// TIA Portal project "Program Monitoring Bearing KAI 2024 (240726)" (V14)

(* hardware
DEVICE "S7-1200 station_1"  S7-1200 Station
   slot 0: "Rack_0"  S7-1200 Rack  Rack  V1.0
   slot 1: "PLC_1"  CPU 1214C DC/DC/DC  6ES7 214-1AG40-0XB0  V4.2
   slot 2: "AI 4x13BIT_1"  6ES7 231-4HD32-0XB0  V2.0
   slot 101: "CP 1243-7 LTE"  CP 1243-7 LTE  6GK7 243-7KX30-0XE0  V3.0
      slot 0: "Telecontrol server"  Partner
      slot 0: "Inter-station communication"  Partner
DEVICE "PC-System_1"  SIMATIC PC station
   slot 0: "SIMATIC PC station"  Rail  SIMATIC PC-Station  V1.0
      slot 125: "Stationmanager"  Station_Manager  V6.0.4
   slot 1: "HMI_RT_1"  WinCC RT Advanced  6AV2 104-0xxxx-xxxx  14.0.1.0
      slot 33792: "Host interface"  Host interface
   slot 2: "IE general_1"  IE General  IE_CP  V8.2.0
*)

// ===== PLC "PLC_1"  CPU 1214C DC/DC/DC =====

VAR_GLOBAL   // PLC tag table "Default tag table"
   "prox_a1" AT %I0.0 : Bool;
   "prox_b1" AT %I0.1 : Bool;
   "Q1-1" AT %M0.0 : Bool;   // utk ngasi trigger biar sensor suhu ngebaca
   "Q2-1" AT %M0.1 : Bool;   // utk ngasi trigger biar sensor suhu ngebaca
   "du_a" AT %M0.2 : Bool;
   "dd_b" AT %M0.3 : Bool;
   "counter" AT %M0.6 : Bool;
   "pemutus" AT %M0.7 : Bool;
   "ProxA+" AT %M1.0 : Bool;
   "ProxB-" AT %M1.1 : Bool;
   "reset" AT %M1.2 : Bool;
   "Clock_Byte" AT %MB10 : Byte;
   "Clock_10Hz" AT %M10.0 : Bool;
   "Clock_5Hz" AT %M10.1 : Bool;
   "Clock_2.5Hz" AT %M10.2 : Bool;
   "Clock_2Hz" AT %M10.3 : Bool;
   "Clock_1.25Hz" AT %M10.4 : Bool;
   "Clock_1Hz" AT %M10.5 : Bool;
   "Clock_0.625Hz" AT %M10.6 : Bool;
   "Clock_0.5Hz" AT %M10.7 : Bool;
   "System_Byte" AT %MB100 : Byte;
   "FirstScan" AT %M100.0 : Bool;
   "DiagStatusUpdate" AT %M100.1 : Bool;
   "AlwaysTRUE" AT %M100.2 : Bool;
   "AlwaysFALSE" AT %M100.3 : Bool;
   "led1" AT %Q0.2 : Bool;
   "led2" AT %Q0.3 : Bool;
   "led3" AT %Q0.4 : Bool;
   "led4" AT %Q0.5 : Bool;
   "led5" AT %Q0.6 : Bool;
   "led6" AT %Q0.7 : Bool;
   "Actual_Step" AT %MW2 : Int;
   "ganjil" AT %M4.0 : Bool;
   "pemutus2" AT %M4.1 : Bool;
   "Q1--2" AT %M2.0 : Bool;   // dipake if nanti sensor suhu ny jd 2 buah (utk datang kanan)
   "Q2-2" AT %M2.1 : Bool;   // dipake if nanti sensor suhu ny jd 2 buah (utk datang kiri)
   "koil timer" AT %M2.4 : Bool;
   "reset koil" AT %M2.3 : Bool;
   "Tag_2" AT %M2.5 : Bool;
   "AI_Sensor Suhu" AT %IW96 : Int;
   "AI_0_Scaled" AT %MD6 : Real;
   "PowerSensorSuhu" AT %Q0.0 : Bool;   // kalo sensor suhu ny jd 2 buah, tambahin satu lg (simpen d network2)
   "Tag_1" AT %M5.0 : Bool;
   "Tag_3" AT %M5.1 : Bool;
   "Tag_4" AT %M5.2 : Bool;
   "Tag_5" AT %M8.0 : Bool;
   "Tag_6" AT %M4.2 : Bool;
   "Tag_7" AT %M9.0 : Bool;
   "Tag_8" AT %M9.3 : Bool;
   "Tag_9" AT %M6.7 : Bool;
   "Tag_10" AT %M12.0 : Bool;
   "Tag_11" AT %MD0 : Time;
   "Tag_12" AT %M8.1 : Bool;
   "Tag_13" AT %M3.0 : Bool;
   "Tag_14" AT %M9.4 : Bool;
   "Tag_15" AT %I0.2 : Bool;
   "Tag_16" AT %M4.4 : Bool;
   "Tag_17" AT %M9.1 : Bool;
   "Tag_18" AT %M9.2 : Bool;
   "Tag_19" AT %M4.3 : Bool;
   "Tag_20" AT %MD2 : DWord;
   "Tag_21" AT %M7.2 : Bool;
   "Tag_22" AT %M3.1 : Bool;
   "Tag_23" AT %M1.3 : Bool;
   "Tag_24" AT %Q1.0 : Bool;
   "Tag_25" AT %M1.4 : Bool;
   "timer_reset" AT %M1.5 : Bool;
   "Suhu_Kanan" AT %MD10 : Real;
   "Tag_27" AT %MD11 : Real;
   "Suhu_Kiri" AT %MD12 : Real;
   "Tag_29" AT %MD13 : Real;
   "Tag_30" AT %MD14 : Real;
   "Tag_31" AT %MD15 : Real;
   "Tag_32" AT %MD16 : Real;
   "Tag_33" AT %MD20 : Real;
   "Tag_34" AT %MD21 : Real;
   "Tag_35" AT %M4.5 : Bool;
   "Tag_36" AT %M4.6 : Bool;
   "Tag_37" AT %M1.6 : Bool;
   "Tag_38" AT %M3.2 : Bool;
   "Tag_39" AT %M3.3 : Bool;
   "Tag_40" AT %M2.2 : Bool;
   "Tag_41" AT %M6.0 : Bool;
   "Tag_42" AT %M6.1 : Bool;
   "Tag_43" AT %M6.2 : Bool;
   "Tag_44" AT %M6.3 : Bool;
   "Tag_45" AT %M6.4 : Bool;
   "Tag_46" AT %M6.5 : Bool;
   "Tag_47" AT %M6.6 : Bool;
   "Tag_48" AT %M7.3 : Bool;
   "Tag_49" AT %M7.4 : Bool;
   "memoryA1" AT %M2.6 : Bool;
   "MemoryB1" AT %M2.7 : Bool;
   "Tag_26" AT %MD1 : Time;
END_VAR

DATA_BLOCK "Data_block_1"   // DB3
{ S7_Optimized_Access := 'FALSE' }
VERSION : 0.1
   VAR
      "counter" : Int;
      "identitas kereta" : String;
      counter_datasuhu : Int := 1;
      sarana : String;
      ganjil : Int := -1;
      genap : Int;
      datasuhu1 : Real;   // Kanan
      datasuhu2 : Real;   // Kiri
      rodakirike : Int;
      rodakananke : Int;
      K1 : Bool;   // Kanan
      K2 : Bool;   // Kiri
      ResetCounterDataSensor : Bool;   // Kanan
      ResetCounterDataSensor1 : Bool;   // Kiri
      ResetCounter100 : Bool;
      Reset : Bool;
      InputKecepatan : Bool;   // Kanan
      InputKecepatan1 : Bool;   // Kiri
      KecepatanKereta : Real;
      Lock_A : Bool;   // Kanan
      Lock_B : Bool;   // Kiri
      ProxB_P : Bool;
      ProxB_N : Bool;
      ProxA_N : Bool;
      ProxA_P : Bool;
      K_B : Bool;
      K_A : Bool;
      WaktuTempuhSensor : Real;
      TimeInput : Bool;
      TimerSensor : Time := T#1ms;
      TimerReset : Time := T#5m;
      datasensor1 : Real;
      datasensor2 : Real;
      data_baru1 : Array[0..99] of Real;   // Kanan
      data_baru2 : Array[0..99] of Real;   // Kiri
      data_suhu_bearing1 : Array[0..99] of Real;
      data_suhu_bearing2 : Array[0..99] of Real;
      data_suhu_bearing3 : Array[0..99] of Real;
      data_suhu_bearing4 : Array[0..99] of Real;
      data_suhu_bearing5 : Array[0..99] of Real;
      data_suhu_bearing6 : Array[0..99] of Real;
      data_suhu_bearing7 : Array[0..99] of Real;
      data_suhu_bearing8 : Array[0..99] of Real;
      data_suhu_bearing9 : Array[0..99] of Real;
      data_suhu_bearing10 : Array[0..99] of Real;
      data_suhu_bearing11 : Array[0..99] of Real;
      data_suhu_bearing12 : Array[0..99] of Real;
      data_suhu_bearing13 : Array[0..99] of Real;
      data_suhu_bearing14 : Array[0..99] of Real;
      data_suhu_bearing15 : Array[0..99] of Real;
      data_suhu_bearing16 : Array[0..99] of Real;
      data_suhu_bearing17 : Array[0..99] of Real;
      data_suhu_bearing18 : Array[0..99] of Real;
      data_suhu_bearing19 : Array[0..99] of Real;
      data_suhu_bearing20 : Array[0..99] of Real;
      data_suhu_bearing21 : Array[0..99] of Real;
      data_suhu_bearing22 : Array[0..99] of Real;
      data_suhu_bearing23 : Array[0..99] of Real;
      data_suhu_bearing24 : Array[0..99] of Real;
      data_suhu_bearing25 : Array[0..99] of Real;
      data_suhu_bearing26 : Array[0..99] of Real;
      data_suhu_bearing27 : Array[0..99] of Real;
      data_suhu_bearing28 : Array[0..99] of Real;
      data_suhu_bearing29 : Array[0..99] of Real;
      data_suhu_bearing30 : Array[0..99] of Real;
      data_suhu_bearing31 : Array[0..99] of Real;
      data_suhu_bearing32 : Array[0..99] of Real;
      data_suhu_bearing33 : Array[0..99] of Real;
      data_suhu_bearing34 : Array[0..99] of Real;
      data_suhu_bearing35 : Array[0..99] of Real;
      data_suhu_bearing36 : Array[0..99] of Real;
      data_suhu_bearing37 : Array[0..99] of Real;
      data_suhu_bearing38 : Array[0..99] of Real;
      data_suhu_bearing39 : Array[0..99] of Real;
      data_suhu_bearing40 : Array[0..99] of Real;
      data_suhu_bearing41 : Array[0..99] of Real;
      data_suhu_bearing42 : Array[0..99] of Real;
      data_suhu_bearing43 : Array[0..99] of Real;
      data_suhu_bearing44 : Array[0..99] of Real;
      data_suhu_bearing45 : Array[0..99] of Real;
      data_suhu_bearing46 : Array[0..99] of Real;
      data_suhu_bearing47 : Array[0..99] of Real;
      data_suhu_bearing48 : Array[0..99] of Real;
      data_suhu_bearing49 : Array[0..99] of Real;
      data_suhu_bearing50 : Array[0..99] of Real;
      data_lama1 : Real;   // Kanan
      data_lama2 : Real;   // Kiri
      dataroda1 : Array[0..49] of Real;   // Kanan
      dataroda2 : Array[0..49] of Real;   // Kiri
      data_0 : Array[0..99] of Real;
      Reset_data_baru1 : Bool;
      counter_sensorA : Int;
      counter_sensorB : Int;
      counterAK1 : Int;
      counterBK1 : Int;
      counterAnotB : Int;
      counterABnot : Int;
      counter_2 : Int;
      counter_1 : Int;
      K10 : Bool;
      counterk1 : Int;
      counterAB : Int;
   END_VAR
BEGIN
END_DATA_BLOCK

// folder: System blocks/Program resources

DATA_BLOCK "IEC_Counter_0_DB_8"   // DB1
{ S7_Optimized_Access := 'TRUE' }
AUTHOR : Simatic
FAMILY : IEC
NAME : CNTR
VERSION : 1.0
// stored: InstanceOfName IEC_COUNTER
"IEC_COUNTER"
BEGIN
END_DATA_BLOCK

DATA_BLOCK "IEC_Timer_0_DB"   // DB2
{ S7_Optimized_Access := 'TRUE' }
AUTHOR : Simatic
FAMILY : IEC
NAME : IEC_TMR
VERSION : 1.0
// stored: InstanceOfName IEC_TIMER
"IEC_TIMER"
BEGIN
END_DATA_BLOCK

DATA_BLOCK "IEC_Counter_0_DB"   // DB4
{ S7_Optimized_Access := 'TRUE' }
AUTHOR : Simatic
FAMILY : IEC
NAME : CNTR
VERSION : 1.0
// stored: InstanceOfName IEC_COUNTER
"IEC_COUNTER"
BEGIN
END_DATA_BLOCK

DATA_BLOCK "IEC_Timer_0_DB_2"   // DB5
{ S7_Optimized_Access := 'TRUE' }
AUTHOR : Simatic
FAMILY : IEC
NAME : IEC_TMR
VERSION : 1.0
// stored: InstanceOfName IEC_TIMER
"IEC_TIMER"
BEGIN
END_DATA_BLOCK

DATA_BLOCK "IEC_Timer_0_DB_1"   // DB6
{ S7_Optimized_Access := 'TRUE' }
AUTHOR : Simatic
FAMILY : IEC
NAME : IEC_TMR
VERSION : 1.0
// stored: InstanceOfName IEC_TIMER
"IEC_TIMER"
BEGIN
END_DATA_BLOCK

DATA_BLOCK "IEC_Timer_0_DB_4"   // DB7
{ S7_Optimized_Access := 'TRUE' }
AUTHOR : Simatic
FAMILY : IEC
NAME : IEC_TMR
VERSION : 1.0
// stored: InstanceOfName IEC_TIMER
"IEC_TIMER"
BEGIN
END_DATA_BLOCK

DATA_BLOCK "IEC_Timer_0_DB_3"   // DB8
{ S7_Optimized_Access := 'TRUE' }
AUTHOR : Simatic
FAMILY : IEC
NAME : IEC_TMR
VERSION : 1.0
// stored: InstanceOfName IEC_TIMER
"IEC_TIMER"
BEGIN
END_DATA_BLOCK

DATA_BLOCK "IEC_Timer_0_DB_5"   // DB9
{ S7_Optimized_Access := 'TRUE' }
AUTHOR : Simatic
FAMILY : IEC
NAME : IEC_TMR
VERSION : 1.0
// stored: InstanceOfName IEC_TIMER
"IEC_TIMER"
BEGIN
END_DATA_BLOCK

DATA_BLOCK "IEC_Counter_0_DB_1"   // DB10
{ S7_Optimized_Access := 'TRUE' }
AUTHOR : Simatic
FAMILY : IEC
NAME : CNTR
VERSION : 1.0
// stored: InstanceOfName IEC_COUNTER
"IEC_COUNTER"
BEGIN
END_DATA_BLOCK

DATA_BLOCK "IEC_Timer_0_DB_7"   // DB11
{ S7_Optimized_Access := 'TRUE' }
AUTHOR : Simatic
FAMILY : IEC
NAME : IEC_TMR
VERSION : 1.0
// stored: InstanceOfName IEC_TIMER
"IEC_TIMER"
BEGIN
END_DATA_BLOCK

DATA_BLOCK "IEC_Timer_0_DB_8"   // DB12
{ S7_Optimized_Access := 'TRUE' }
AUTHOR : Simatic
FAMILY : IEC
NAME : IEC_TMR
VERSION : 1.0
// stored: InstanceOfName IEC_TIMER
"IEC_TIMER"
BEGIN
END_DATA_BLOCK

DATA_BLOCK "IEC_Timer_0_DB_9"   // DB13
{ S7_Optimized_Access := 'TRUE' }
AUTHOR : Simatic
FAMILY : IEC
NAME : IEC_TMR
VERSION : 1.0
// stored: InstanceOfName IEC_TIMER
"IEC_TIMER"
BEGIN
END_DATA_BLOCK

DATA_BLOCK "IEC_Timer_0_DB_10"   // DB14
{ S7_Optimized_Access := 'TRUE' }
AUTHOR : Simatic
FAMILY : IEC
NAME : IEC_TMR
VERSION : 1.0
// stored: InstanceOfName IEC_TIMER
"IEC_TIMER"
BEGIN
END_DATA_BLOCK

DATA_BLOCK "IEC_Timer_0_DB_11"   // DB15
{ S7_Optimized_Access := 'TRUE' }
AUTHOR : Simatic
FAMILY : IEC
NAME : IEC_TMR
VERSION : 1.0
// stored: InstanceOfName IEC_TIMER
"IEC_TIMER"
BEGIN
END_DATA_BLOCK

DATA_BLOCK "IEC_Counter_0_DB_2"   // DB17
{ S7_Optimized_Access := 'TRUE' }
AUTHOR : Simatic
FAMILY : IEC
NAME : CNTR
VERSION : 1.0
// stored: InstanceOfName IEC_COUNTER
"IEC_COUNTER"
BEGIN
END_DATA_BLOCK

DATA_BLOCK "IEC_Counter_0_DB_3"   // DB18
{ S7_Optimized_Access := 'TRUE' }
AUTHOR : Simatic
FAMILY : IEC
NAME : CNTR
VERSION : 1.0
// stored: InstanceOfName IEC_COUNTER
"IEC_COUNTER"
BEGIN
END_DATA_BLOCK

DATA_BLOCK "IEC_Counter_0_DB_4"   // DB19
{ S7_Optimized_Access := 'TRUE' }
AUTHOR : Simatic
FAMILY : IEC
NAME : CNTR
VERSION : 1.0
// stored: InstanceOfName IEC_COUNTER
"IEC_COUNTER"
BEGIN
END_DATA_BLOCK

DATA_BLOCK "IEC_Counter_0_DB_5"   // DB20
{ S7_Optimized_Access := 'TRUE' }
AUTHOR : Simatic
FAMILY : IEC
NAME : CNTR
VERSION : 1.0
// stored: InstanceOfName IEC_COUNTER
"IEC_COUNTER"
BEGIN
END_DATA_BLOCK

DATA_BLOCK "IEC_Counter_0_DB_6"   // DB21
{ S7_Optimized_Access := 'TRUE' }
AUTHOR : Simatic
FAMILY : IEC
NAME : CNTR
VERSION : 1.0
// stored: InstanceOfName IEC_COUNTER
"IEC_COUNTER"
BEGIN
END_DATA_BLOCK

DATA_BLOCK "IEC_Counter_0_DB_7"   // DB22
{ S7_Optimized_Access := 'TRUE' }
AUTHOR : Simatic
FAMILY : IEC
NAME : CNTR
VERSION : 1.0
// stored: InstanceOfName IEC_COUNTER
"IEC_COUNTER"
BEGIN
END_DATA_BLOCK

DATA_BLOCK "IEC_Counter_0_DB_11"   // DB23
{ S7_Optimized_Access := 'TRUE' }
AUTHOR : Simatic
FAMILY : IEC
NAME : CNTR
VERSION : 1.0
// stored: InstanceOfName IEC_COUNTER
"IEC_COUNTER"
BEGIN
END_DATA_BLOCK

DATA_BLOCK "IEC_Timer_0_DB_6"   // DB24
{ S7_Optimized_Access := 'TRUE' }
AUTHOR : Simatic
FAMILY : IEC
NAME : IEC_TMR
VERSION : 1.0
// stored: InstanceOfName IEC_TIMER
"IEC_TIMER"
BEGIN
END_DATA_BLOCK

DATA_BLOCK "IEC_Timer_0_DB_12"   // DB25
{ S7_Optimized_Access := 'TRUE' }
AUTHOR : Simatic
FAMILY : IEC
NAME : IEC_TMR
VERSION : 1.0
// stored: InstanceOfName IEC_TIMER
"IEC_TIMER"
BEGIN
END_DATA_BLOCK

// folder: (top level)

FUNCTION "Block_1" : Void   // FC1, LAD
{ S7_Optimized_Access := 'TRUE' }
VERSION : 0.1
   VAR_INPUT
      "analog input suhu" : Int;
      lower : Real;
      upper : Real;
   END_VAR
   VAR_OUTPUT
      "Scaled Output Suhu" : Real;
   END_VAR
   VAR_TEMP
      Temp1 : Real;   // temporary data
   END_VAR
BEGIN

REGION Network 1
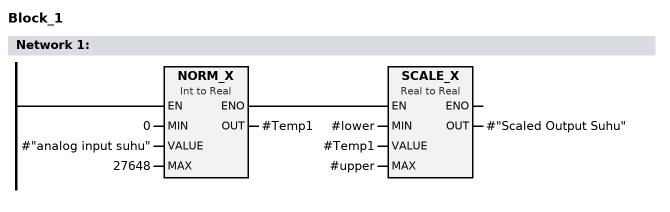
   RUNG wire#powerrail
      { S7_Templates := "[SrcType := Int, DestType := Real]" } Normalize(min := 0, value := #"analog input suhu", max := 27648, out => #Temp1)
      { S7_Templates := "[SrcType := Real, DestType := Real]" } Scale(min := #lower, value := #Temp1, max := #upper, out => #"Scaled Output Suhu")
   END_RUNG
   // the same network as SCL:
   #Temp1 := NORM_X(MIN := 0, VALUE := #"analog input suhu", MAX := 27648);
   #"Scaled Output Suhu" := SCALE_X(MIN := #lower, VALUE := #Temp1, MAX := #upper);
END_REGION
END_FUNCTION

ORGANIZATION_BLOCK "Program Datang Kiri"   // OB1, LAD, ProgramCycle
TITLE = Datang Kiri
{ S7_Optimized_Access := 'TRUE' }
VERSION : 0.1
   VAR_INPUT
      Initial_Call : Bool;   // Initial call of this OB
      Remanence : Bool;   // =True, if remanent data are available
   END_VAR
   VAR CONSTANT
      initial_step : Int;
      step_led1 : Int := 1;
      step_led2 : Int := 2;
      step_led3 : Int := 3;
      step_led4 : Int := 4;
      step_led5 : Int := 5;
      step_led6 : Int := 6;
   END_VAR
   VAR_TEMP   // added for the SCL form of the ladder/FBD networks
      _w1 : Bool;
      _w2 : Bool;
      _w3 : Bool;
      _w4 : Bool;
      _w5 : Bool;
      _w6 : Bool;
      _w7 : Bool;
      _w8 : Bool;
      _w9 : Bool;
      _w10 : Bool;
      _w11 : Bool;
      _w12 : Bool;
      _w13 : Bool;
      _w14 : Bool;
      _w15 : Bool;
      _w16 : Bool;
      _w17 : Bool;
      _w18 : Bool;
      _w19 : Bool;
      _w20 : Bool;
      _w21 : Bool;
      _w22 : Bool;
      _w23 : Bool;
      _w24 : Bool;
      _w25 : Bool;
      _w26 : Bool;
      _w27 : Bool;
      _w28 : Bool;
      _w29 : Bool;
      _w30 : Bool;
      _w31 : Bool;
      _w32 : Bool;
      _w33 : Bool;
      _w34 : Bool;
      _w35 : Bool;
      _w36 : Bool;
      _w37 : Bool;
      _w38 : Bool;
      _w39 : Bool;
      _w40 : Bool;
      _w41 : Bool;
      _w42 : Bool;
      _w43 : Bool;
      _w44 : Bool;
      _w45 : Bool;
      _w46 : Bool;
      _w47 : Bool;
      _w48 : Bool;
      _w49 : Bool;
      _w50 : Bool;
   END_VAR
BEGIN

REGION Network 1: Koil Mengukur kecepatan kereta (kiri ke kanan)
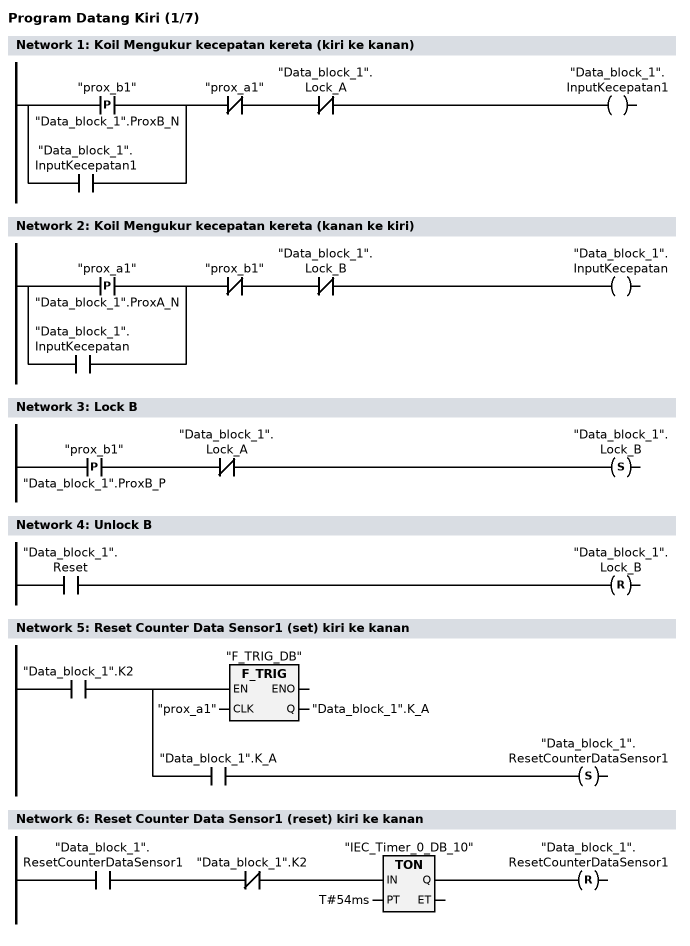
   RUNG wire#powerrail
      P_Contact(operand := "prox_b1", bit := "Data_block_1".ProxB_N)
      wire#w1
      I_Contact( "prox_a1" )
      I_Contact( "Data_block_1".Lock_A )
      Coil( "Data_block_1".InputKecepatan1 )
   END_RUNG
   RUNG wire#powerrail
      Contact( "Data_block_1".InputKecepatan1 )
   END_RUNG wire#w1
   // the same network as SCL:
   #_w1 := "prox_b1" AND NOT "Data_block_1".ProxB_N;   // rising edge of "prox_b1"
   "Data_block_1".ProxB_N := "prox_b1";
   "Data_block_1".InputKecepatan1 := (#_w1 OR "Data_block_1".InputKecepatan1) AND NOT "prox_a1" AND NOT "Data_block_1".Lock_A;
END_REGION

REGION Network 2: Koil Mengukur kecepatan kereta (kanan ke kiri)
   RUNG wire#powerrail
      P_Contact(operand := "prox_a1", bit := "Data_block_1".ProxA_N)
      wire#w1
      I_Contact( "prox_b1" )
      I_Contact( "Data_block_1".Lock_B )
      Coil( "Data_block_1".InputKecepatan )
   END_RUNG
   RUNG wire#powerrail
      Contact( "Data_block_1".InputKecepatan )
   END_RUNG wire#w1
   // the same network as SCL:
   #_w1 := "prox_a1" AND NOT "Data_block_1".ProxA_N;   // rising edge of "prox_a1"
   "Data_block_1".ProxA_N := "prox_a1";
   "Data_block_1".InputKecepatan := (#_w1 OR "Data_block_1".InputKecepatan) AND NOT "prox_b1" AND NOT "Data_block_1".Lock_B;
END_REGION

REGION Network 3: Lock B
   RUNG wire#powerrail
      P_Contact(operand := "prox_b1", bit := "Data_block_1".ProxB_P)
      I_Contact( "Data_block_1".Lock_A )
      S_Coil( "Data_block_1".Lock_B )
   END_RUNG
   // the same network as SCL:
   #_w1 := "prox_b1" AND NOT "Data_block_1".ProxB_P;   // rising edge of "prox_b1"
   "Data_block_1".ProxB_P := "prox_b1";
   IF #_w1 AND NOT "Data_block_1".Lock_A THEN "Data_block_1".Lock_B := TRUE; END_IF;
END_REGION

REGION Network 4: Unlock B
   RUNG wire#powerrail
      Contact( "Data_block_1".Reset )
      R_Coil( "Data_block_1".Lock_B )
   END_RUNG
   // the same network as SCL:
   IF "Data_block_1".Reset THEN "Data_block_1".Lock_B := FALSE; END_IF;
END_REGION

REGION Network 5: Reset Counter Data Sensor1 (set) kiri ke kanan
   IF "Data_block_1".K2 THEN
       "F_TRIG_DB"(CLK := "prox_a1", Q => "Data_block_1".K_A);   // F_TRIG
   END_IF;
   IF "Data_block_1".K2 AND "Data_block_1".K_A THEN "Data_block_1".ResetCounterDataSensor1 := TRUE; END_IF;
END_REGION

REGION Network 6: Reset Counter Data Sensor1 (reset) kiri ke kanan
   "IEC_Timer_0_DB_10".TON(IN := "Data_block_1".ResetCounterDataSensor1 AND NOT "Data_block_1".K2, PT := T#54ms);
   IF "IEC_Timer_0_DB_10".Q THEN "Data_block_1".ResetCounterDataSensor1 := FALSE; END_IF;
END_REGION

REGION Network 7: reset data_baru (kiri ke kanan) data_baru2
   // ketika reset aktif 
   // 
   // - maka datasuhu, array data suhu roda akan kembali 0
   // - maka counter genap kembali 0
   // - maka counter ganjil menjadi -1
   // - maka sarana akan kosong
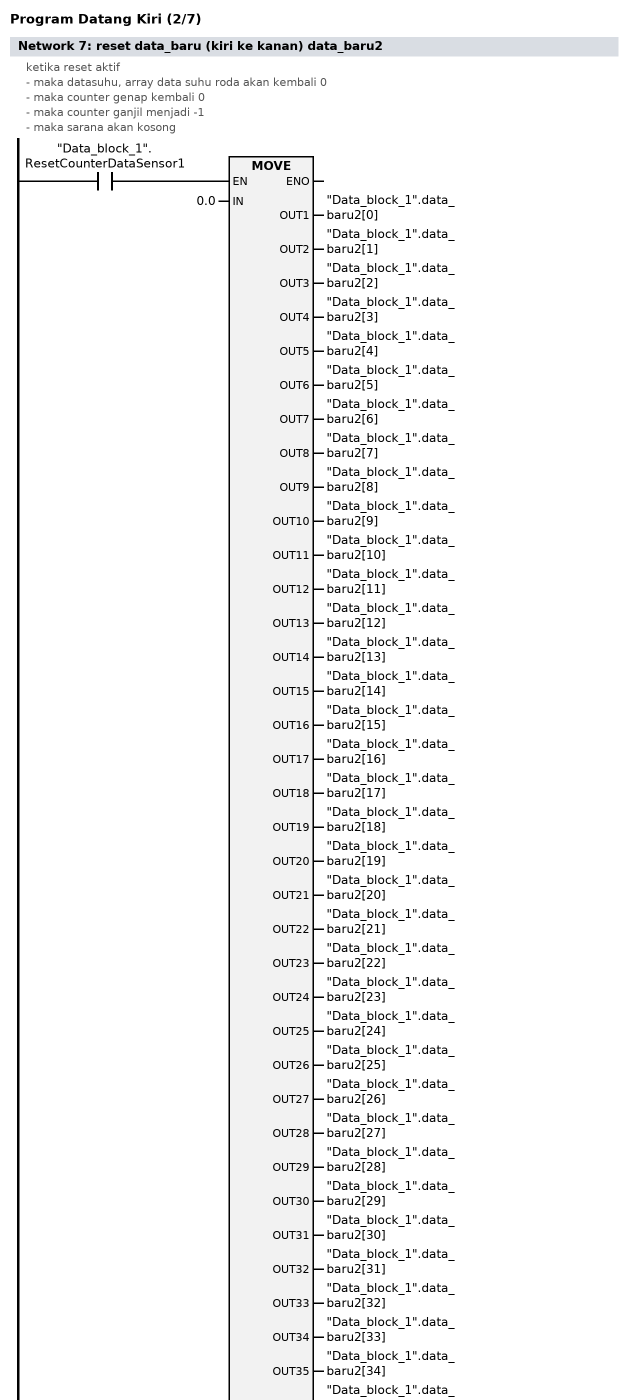
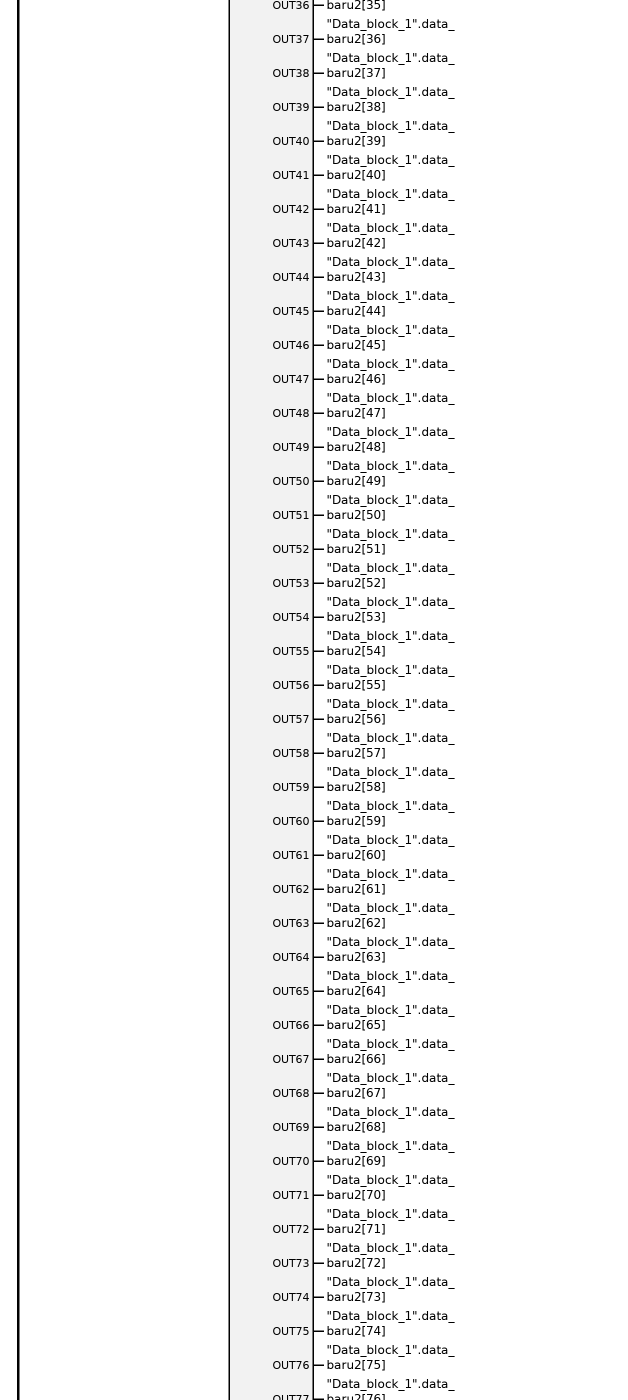
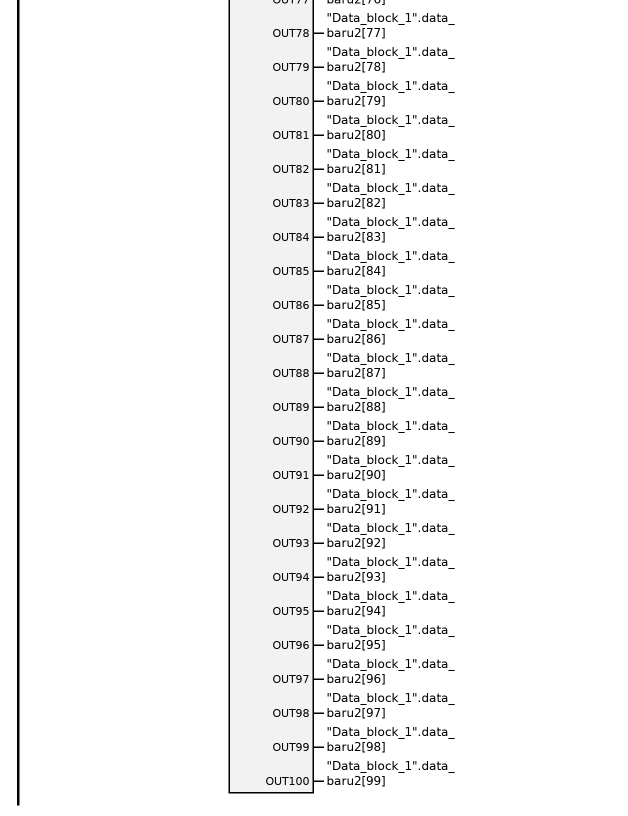
   RUNG wire#powerrail
      Contact( "Data_block_1".ResetCounterDataSensor1 )
      Move(in := 0.0, out1 => "Data_block_1".data_baru2[0], out2 => "Data_block_1".data_baru2[1], out3 => "Data_block_1".data_baru2[2], out4 => "Data_block_1".data_baru2[3], out5 => "Data_block_1".data_baru2[4], out6 => "Data_block_1".data_baru2[5], out7 => "Data_block_1".data_baru2[6], out8 => "Data_block_1".data_baru2[7], out9 => "Data_block_1".data_baru2[8], out10 => "Data_block_1".data_baru2[9], out11 => "Data_block_1".data_baru2[10], out12 => "Data_block_1".data_baru2[11], out13 => "Data_block_1".data_baru2[12], out14 => "Data_block_1".data_baru2[13], out15 => "Data_block_1".data_baru2[14], out16 => "Data_block_1".data_baru2[15], out17 => "Data_block_1".data_baru2[16], out18 => "Data_block_1".data_baru2[17], out19 => "Data_block_1".data_baru2[18], out20 => "Data_block_1".data_baru2[19], out21 => "Data_block_1".data_baru2[20], out22 => "Data_block_1".data_baru2[21], out23 => "Data_block_1".data_baru2[22], out24 => "Data_block_1".data_baru2[23], out25 => "Data_block_1".data_baru2[24], out26 => "Data_block_1".data_baru2[25], out27 => "Data_block_1".data_baru2[26], out28 => "Data_block_1".data_baru2[27], out29 => "Data_block_1".data_baru2[28], out30 => "Data_block_1".data_baru2[29], out31 => "Data_block_1".data_baru2[30], out32 => "Data_block_1".data_baru2[31], out33 => "Data_block_1".data_baru2[32], out34 => "Data_block_1".data_baru2[33], out35 => "Data_block_1".data_baru2[34], out36 => "Data_block_1".data_baru2[35], out37 => "Data_block_1".data_baru2[36], out38 => "Data_block_1".data_baru2[37], out39 => "Data_block_1".data_baru2[38], out40 => "Data_block_1".data_baru2[39], out41 => "Data_block_1".data_baru2[40], out42 => "Data_block_1".data_baru2[41], out43 => "Data_block_1".data_baru2[42], out44 => "Data_block_1".data_baru2[43], out45 => "Data_block_1".data_baru2[44], out46 => "Data_block_1".data_baru2[45], out47 => "Data_block_1".data_baru2[46], out48 => "Data_block_1".data_baru2[47], out49 => "Data_block_1".data_baru2[48], out50 => "Data_block_1".data_baru2[49], out51 => "Data_block_1".data_baru2[50], out52 => "Data_block_1".data_baru2[51], out53 => "Data_block_1".data_baru2[52], out54 => "Data_block_1".data_baru2[53], out55 => "Data_block_1".data_baru2[54], out56 => "Data_block_1".data_baru2[55], out57 => "Data_block_1".data_baru2[56], out58 => "Data_block_1".data_baru2[57], out59 => "Data_block_1".data_baru2[58], out60 => "Data_block_1".data_baru2[59], out61 => "Data_block_1".data_baru2[60], out62 => "Data_block_1".data_baru2[61], out63 => "Data_block_1".data_baru2[62], out64 => "Data_block_1".data_baru2[63], out65 => "Data_block_1".data_baru2[64], out66 => "Data_block_1".data_baru2[65], out67 => "Data_block_1".data_baru2[66], out68 => "Data_block_1".data_baru2[67], out69 => "Data_block_1".data_baru2[68], out70 => "Data_block_1".data_baru2[69], out71 => "Data_block_1".data_baru2[70], out72 => "Data_block_1".data_baru2[71], out73 => "Data_block_1".data_baru2[72], out74 => "Data_block_1".data_baru2[73], out75 => "Data_block_1".data_baru2[74], out76 => "Data_block_1".data_baru2[75], out77 => "Data_block_1".data_baru2[76], out78 => "Data_block_1".data_baru2[77], out79 => "Data_block_1".data_baru2[78], out80 => "Data_block_1".data_baru2[79], out81 => "Data_block_1".data_baru2[80], out82 => "Data_block_1".data_baru2[81], out83 => "Data_block_1".data_baru2[82], out84 => "Data_block_1".data_baru2[83], out85 => "Data_block_1".data_baru2[84], out86 => "Data_block_1".data_baru2[85], out87 => "Data_block_1".data_baru2[86], out88 => "Data_block_1".data_baru2[87], out89 => "Data_block_1".data_baru2[88], out90 => "Data_block_1".data_baru2[89], out91 => "Data_block_1".data_baru2[90], out92 => "Data_block_1".data_baru2[91], out93 => "Data_block_1".data_baru2[92], out94 => "Data_block_1".data_baru2[93], out95 => "Data_block_1".data_baru2[94], out96 => "Data_block_1".data_baru2[95], out97 => "Data_block_1".data_baru2[96], out98 => "Data_block_1".data_baru2[97], out99 => "Data_block_1".data_baru2[98], out100 => "Data_block_1".data_baru2[99])
   END_RUNG
   // the same network as SCL:
   IF "Data_block_1".ResetCounterDataSensor1 THEN
       "Data_block_1".data_baru2[0] := 0.0;
       "Data_block_1".data_baru2[1] := 0.0;
       "Data_block_1".data_baru2[2] := 0.0;
       "Data_block_1".data_baru2[3] := 0.0;
       "Data_block_1".data_baru2[4] := 0.0;
       "Data_block_1".data_baru2[5] := 0.0;
       "Data_block_1".data_baru2[6] := 0.0;
       "Data_block_1".data_baru2[7] := 0.0;
       "Data_block_1".data_baru2[8] := 0.0;
       "Data_block_1".data_baru2[9] := 0.0;
       "Data_block_1".data_baru2[10] := 0.0;
       "Data_block_1".data_baru2[11] := 0.0;
       "Data_block_1".data_baru2[12] := 0.0;
       "Data_block_1".data_baru2[13] := 0.0;
       "Data_block_1".data_baru2[14] := 0.0;
       "Data_block_1".data_baru2[15] := 0.0;
       "Data_block_1".data_baru2[16] := 0.0;
       "Data_block_1".data_baru2[17] := 0.0;
       "Data_block_1".data_baru2[18] := 0.0;
       "Data_block_1".data_baru2[19] := 0.0;
       "Data_block_1".data_baru2[20] := 0.0;
       "Data_block_1".data_baru2[21] := 0.0;
       "Data_block_1".data_baru2[22] := 0.0;
       "Data_block_1".data_baru2[23] := 0.0;
       "Data_block_1".data_baru2[24] := 0.0;
       "Data_block_1".data_baru2[25] := 0.0;
       "Data_block_1".data_baru2[26] := 0.0;
       "Data_block_1".data_baru2[27] := 0.0;
       "Data_block_1".data_baru2[28] := 0.0;
       "Data_block_1".data_baru2[29] := 0.0;
       "Data_block_1".data_baru2[30] := 0.0;
       "Data_block_1".data_baru2[31] := 0.0;
       "Data_block_1".data_baru2[32] := 0.0;
       "Data_block_1".data_baru2[33] := 0.0;
       "Data_block_1".data_baru2[34] := 0.0;
       "Data_block_1".data_baru2[35] := 0.0;
       "Data_block_1".data_baru2[36] := 0.0;
       "Data_block_1".data_baru2[37] := 0.0;
       "Data_block_1".data_baru2[38] := 0.0;
       "Data_block_1".data_baru2[39] := 0.0;
       "Data_block_1".data_baru2[40] := 0.0;
       "Data_block_1".data_baru2[41] := 0.0;
       "Data_block_1".data_baru2[42] := 0.0;
       "Data_block_1".data_baru2[43] := 0.0;
       "Data_block_1".data_baru2[44] := 0.0;
       "Data_block_1".data_baru2[45] := 0.0;
       "Data_block_1".data_baru2[46] := 0.0;
       "Data_block_1".data_baru2[47] := 0.0;
       "Data_block_1".data_baru2[48] := 0.0;
       "Data_block_1".data_baru2[49] := 0.0;
       "Data_block_1".data_baru2[50] := 0.0;
       "Data_block_1".data_baru2[51] := 0.0;
       "Data_block_1".data_baru2[52] := 0.0;
       "Data_block_1".data_baru2[53] := 0.0;
       "Data_block_1".data_baru2[54] := 0.0;
       "Data_block_1".data_baru2[55] := 0.0;
       "Data_block_1".data_baru2[56] := 0.0;
       "Data_block_1".data_baru2[57] := 0.0;
       "Data_block_1".data_baru2[58] := 0.0;
       "Data_block_1".data_baru2[59] := 0.0;
       "Data_block_1".data_baru2[60] := 0.0;
       "Data_block_1".data_baru2[61] := 0.0;
       "Data_block_1".data_baru2[62] := 0.0;
       "Data_block_1".data_baru2[63] := 0.0;
       "Data_block_1".data_baru2[64] := 0.0;
       "Data_block_1".data_baru2[65] := 0.0;
       "Data_block_1".data_baru2[66] := 0.0;
       "Data_block_1".data_baru2[67] := 0.0;
       "Data_block_1".data_baru2[68] := 0.0;
       "Data_block_1".data_baru2[69] := 0.0;
       "Data_block_1".data_baru2[70] := 0.0;
       "Data_block_1".data_baru2[71] := 0.0;
       "Data_block_1".data_baru2[72] := 0.0;
       "Data_block_1".data_baru2[73] := 0.0;
       "Data_block_1".data_baru2[74] := 0.0;
       "Data_block_1".data_baru2[75] := 0.0;
       "Data_block_1".data_baru2[76] := 0.0;
       "Data_block_1".data_baru2[77] := 0.0;
       "Data_block_1".data_baru2[78] := 0.0;
       "Data_block_1".data_baru2[79] := 0.0;
       "Data_block_1".data_baru2[80] := 0.0;
       "Data_block_1".data_baru2[81] := 0.0;
       "Data_block_1".data_baru2[82] := 0.0;
       "Data_block_1".data_baru2[83] := 0.0;
       "Data_block_1".data_baru2[84] := 0.0;
       "Data_block_1".data_baru2[85] := 0.0;
       "Data_block_1".data_baru2[86] := 0.0;
       "Data_block_1".data_baru2[87] := 0.0;
       "Data_block_1".data_baru2[88] := 0.0;
       "Data_block_1".data_baru2[89] := 0.0;
       "Data_block_1".data_baru2[90] := 0.0;
       "Data_block_1".data_baru2[91] := 0.0;
       "Data_block_1".data_baru2[92] := 0.0;
       "Data_block_1".data_baru2[93] := 0.0;
       "Data_block_1".data_baru2[94] := 0.0;
       "Data_block_1".data_baru2[95] := 0.0;
       "Data_block_1".data_baru2[96] := 0.0;
       "Data_block_1".data_baru2[97] := 0.0;
       "Data_block_1".data_baru2[98] := 0.0;
       "Data_block_1".data_baru2[99] := 0.0;
   END_IF;
END_REGION

REGION Network 8: Koil Set Proxy B (kiri ke kanan)
   // Sensor A aktif, menunjukkan arah kereta dari arah kanan
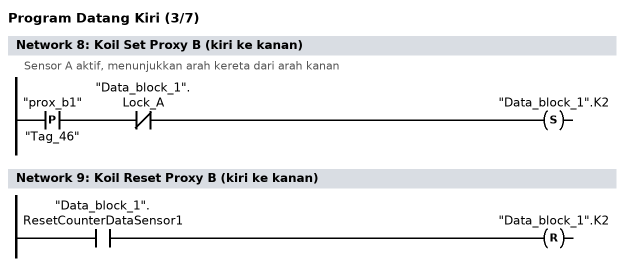
   RUNG wire#powerrail
      P_Contact(operand := "prox_b1", bit := "Tag_46")
      I_Contact( "Data_block_1".Lock_A )
      S_Coil( "Data_block_1".K2 )
   END_RUNG
   // the same network as SCL:
   #_w1 := "prox_b1" AND NOT "Tag_46";   // rising edge of "prox_b1"
   "Tag_46" := "prox_b1";
   IF #_w1 AND NOT "Data_block_1".Lock_A THEN "Data_block_1".K2 := TRUE; END_IF;
END_REGION

REGION Network 9: Koil Reset Proxy B (kiri ke kanan)
   RUNG wire#powerrail
      Contact( "Data_block_1".ResetCounterDataSensor1 )
      R_Coil( "Data_block_1".K2 )
   END_RUNG
   // the same network as SCL:
   IF "Data_block_1".ResetCounterDataSensor1 THEN "Data_block_1".K2 := FALSE; END_IF;
END_REGION

REGION Network 10: Mengukur Suhu Roda (kiri ke kanan)
   // setelah sensor suhu aktif membaca
   // kemudian counter menghitung jumlah berapa kali sensor suhu mendeteksi suhu pada satu roda
   // 
   // apabila data sensor suhu yang terbaca(datasensor) tidak sama dengan nol maka data suhu yang terbaca(datasensor) dipindahkan ke array data suhu baru (data_baru1 untuk sebelah kanan) (data_baru2 untuk sebelah kiri)
   // data sensor terbaru dirubah jadi data baru
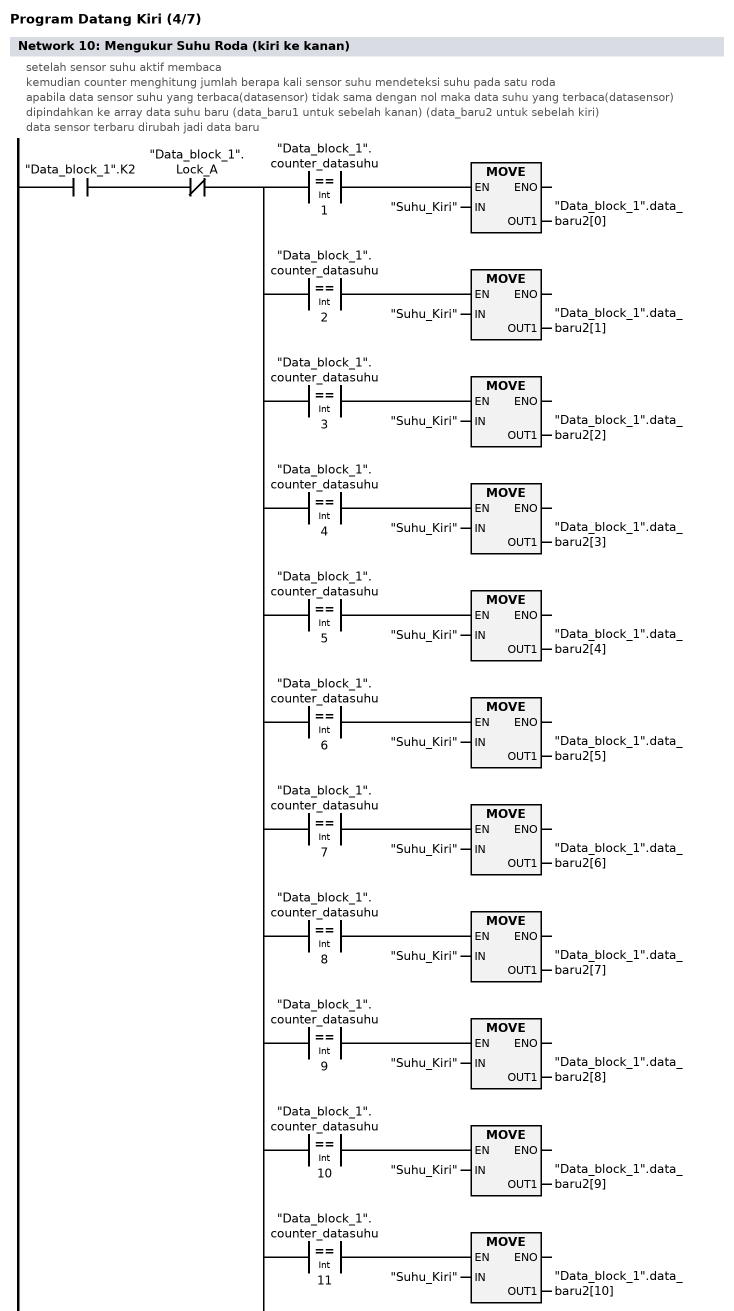
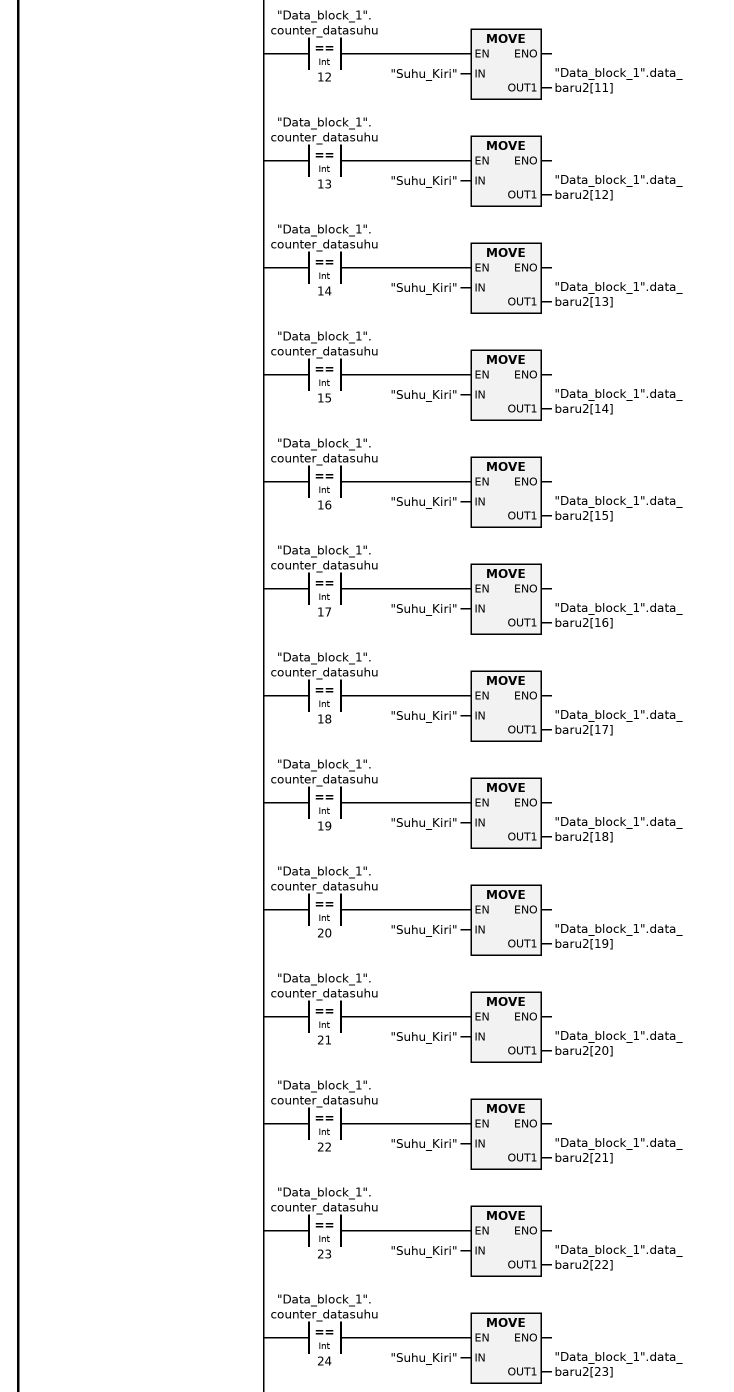
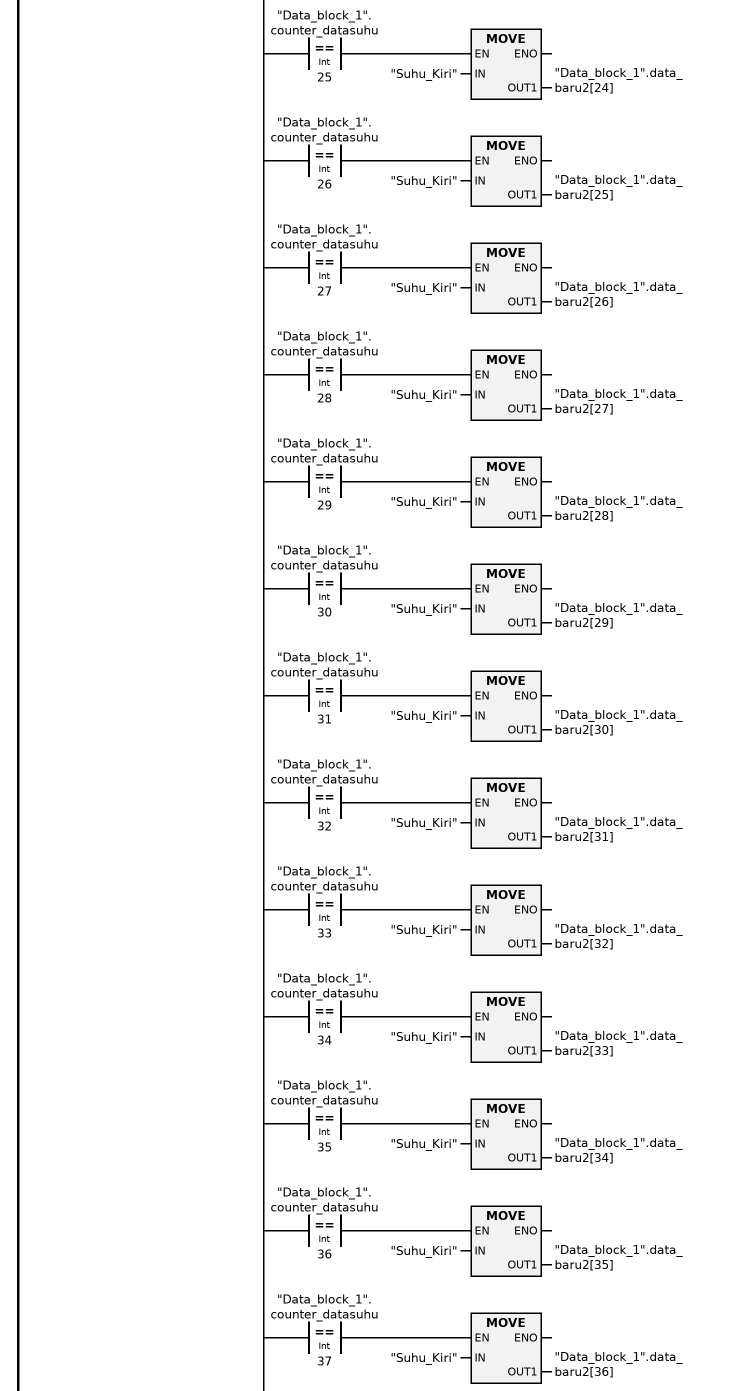
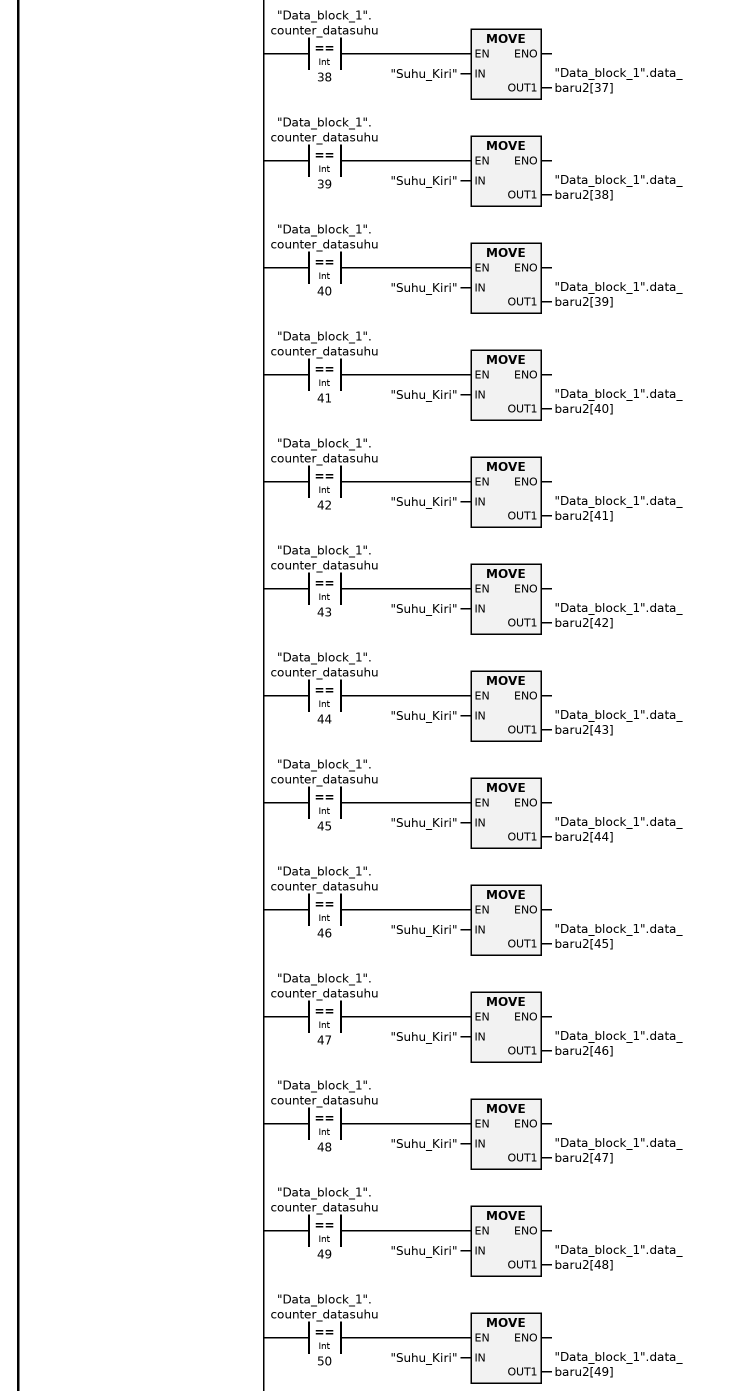
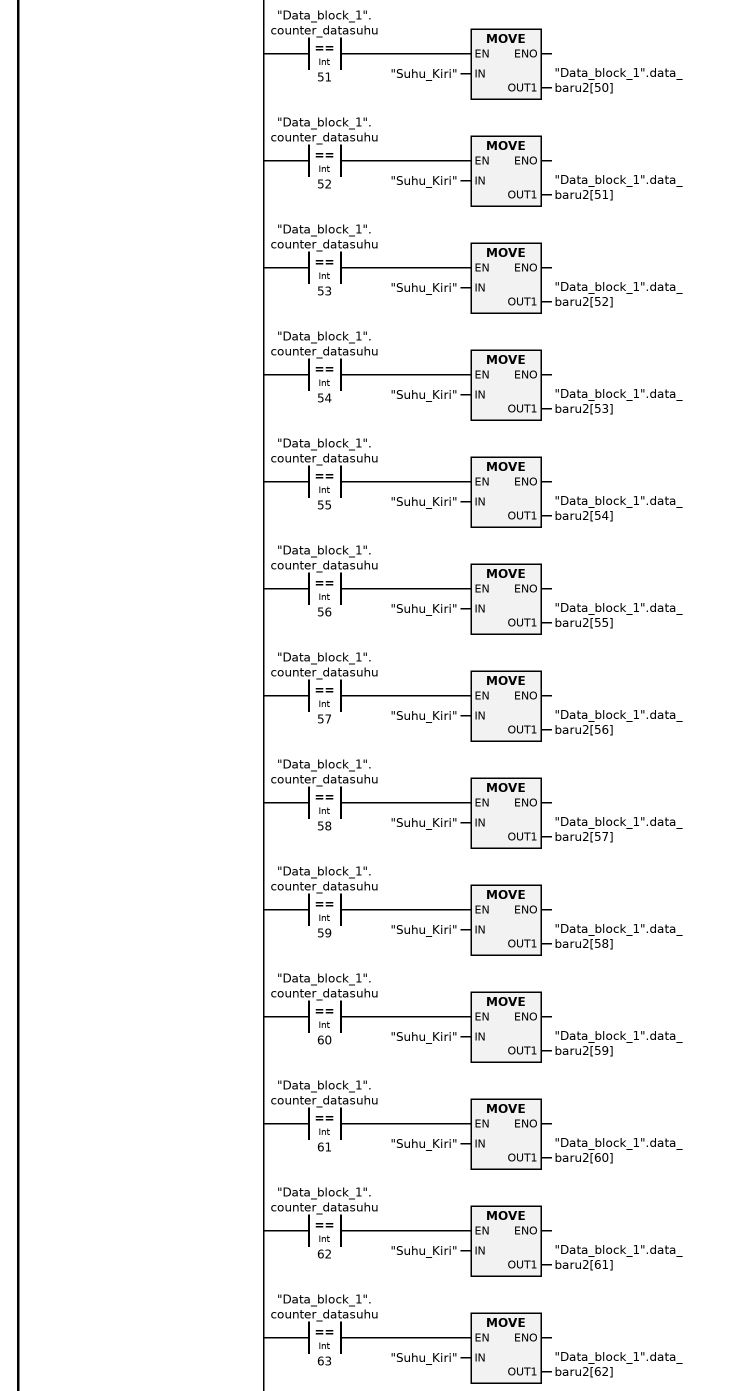
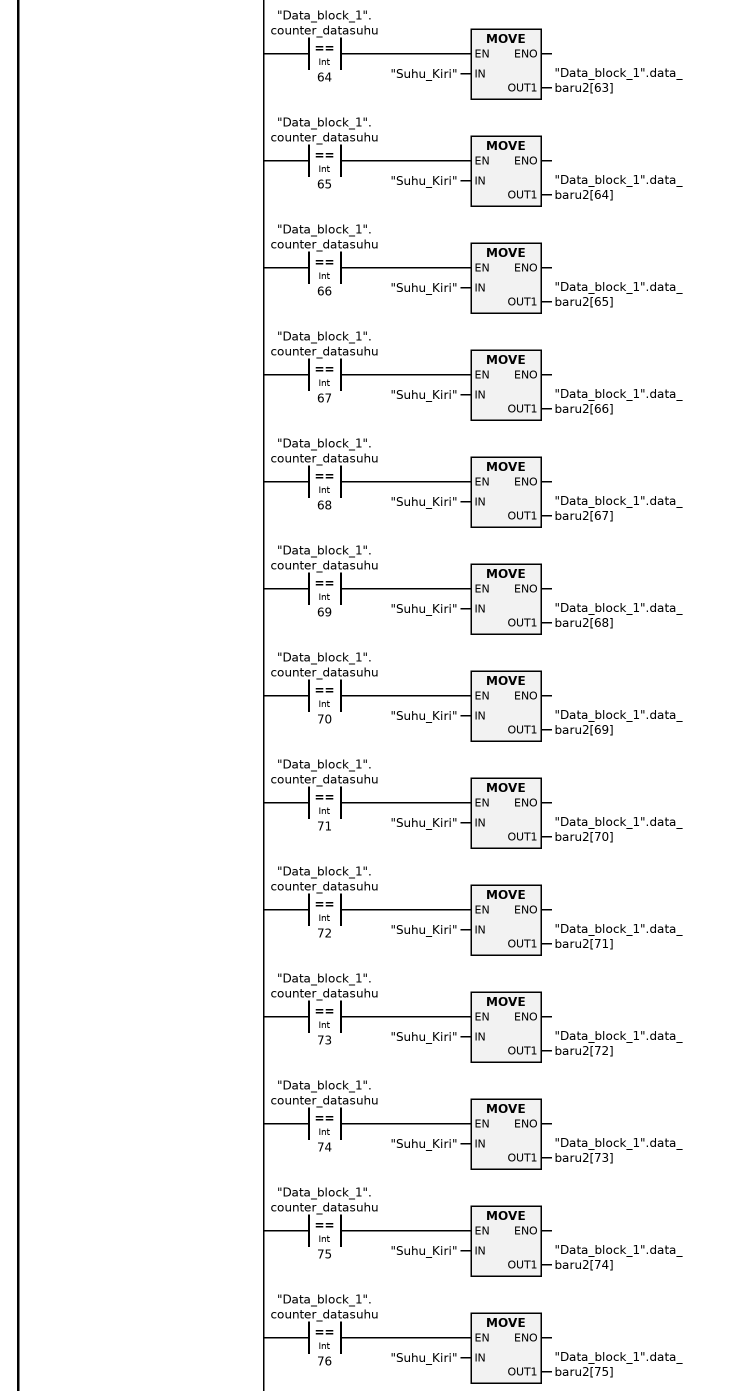
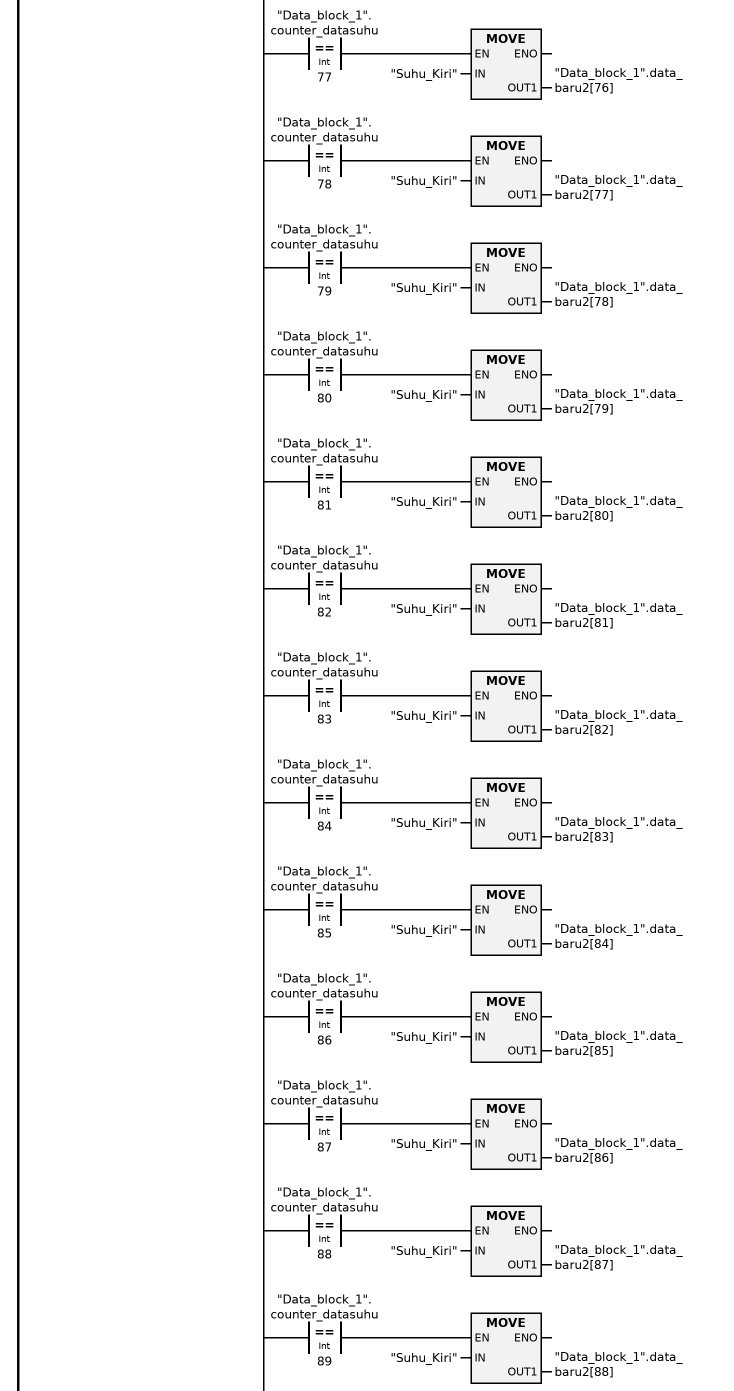
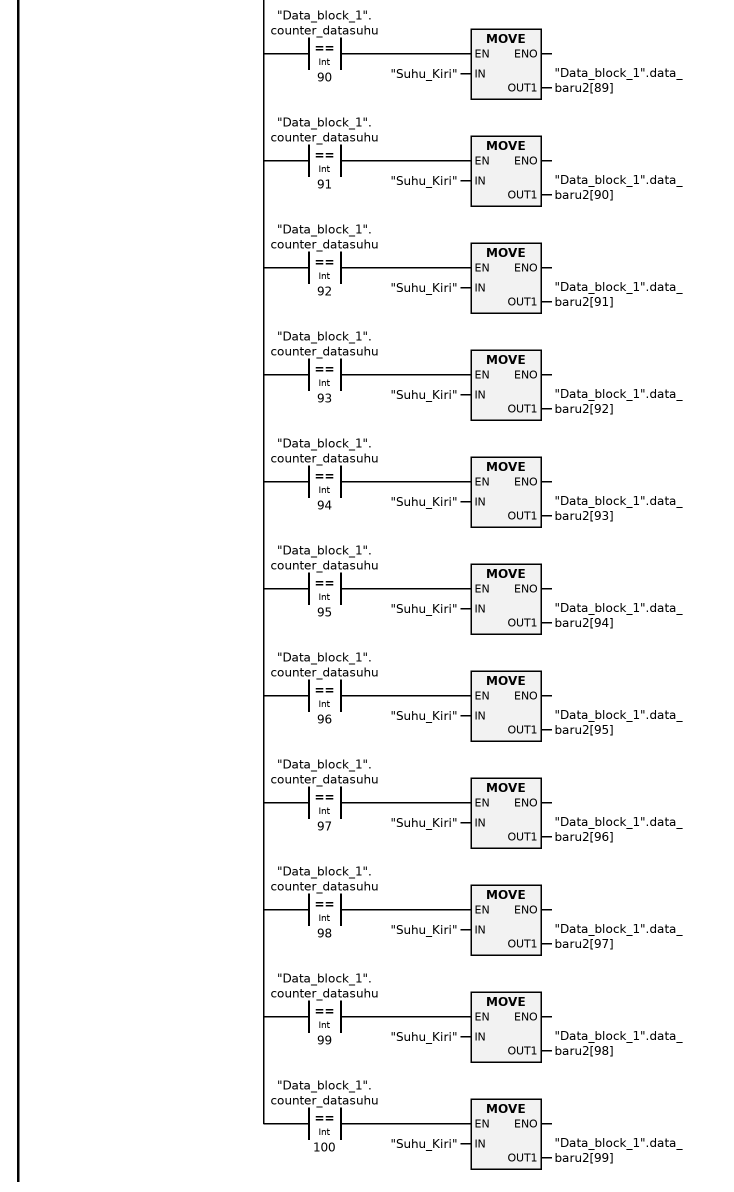
   RUNG wire#powerrail
      Contact( "Data_block_1".K2 )
      I_Contact( "Data_block_1".Lock_A )
      wire#w1
      { S7_Templates := "SrcType := Int" } EQ_Contact(in1 := "Data_block_1".counter_datasuhu, in2 := 1)
      Move(in := "Suhu_Kiri", out1 => "Data_block_1".data_baru2[0])
   END_RUNG
   RUNG wire#w1
      { S7_Templates := "SrcType := Int" } EQ_Contact(in1 := "Data_block_1".counter_datasuhu, in2 := 2)
      Move(in := "Suhu_Kiri", out1 => "Data_block_1".data_baru2[1])
   END_RUNG
   RUNG wire#w1
      { S7_Templates := "SrcType := Int" } EQ_Contact(in1 := "Data_block_1".counter_datasuhu, in2 := 3)
      Move(in := "Suhu_Kiri", out1 => "Data_block_1".data_baru2[2])
   END_RUNG
   RUNG wire#w1
      { S7_Templates := "SrcType := Int" } EQ_Contact(in1 := "Data_block_1".counter_datasuhu, in2 := 4)
      Move(in := "Suhu_Kiri", out1 => "Data_block_1".data_baru2[3])
   END_RUNG
   RUNG wire#w1
      { S7_Templates := "SrcType := Int" } EQ_Contact(in1 := "Data_block_1".counter_datasuhu, in2 := 5)
      Move(in := "Suhu_Kiri", out1 => "Data_block_1".data_baru2[4])
   END_RUNG
   RUNG wire#w1
      { S7_Templates := "SrcType := Int" } EQ_Contact(in1 := "Data_block_1".counter_datasuhu, in2 := 6)
      Move(in := "Suhu_Kiri", out1 => "Data_block_1".data_baru2[5])
   END_RUNG
   RUNG wire#w1
      { S7_Templates := "SrcType := Int" } EQ_Contact(in1 := "Data_block_1".counter_datasuhu, in2 := 7)
      Move(in := "Suhu_Kiri", out1 => "Data_block_1".data_baru2[6])
   END_RUNG
   RUNG wire#w1
      { S7_Templates := "SrcType := Int" } EQ_Contact(in1 := "Data_block_1".counter_datasuhu, in2 := 8)
      Move(in := "Suhu_Kiri", out1 => "Data_block_1".data_baru2[7])
   END_RUNG
   RUNG wire#w1
      { S7_Templates := "SrcType := Int" } EQ_Contact(in1 := "Data_block_1".counter_datasuhu, in2 := 9)
      Move(in := "Suhu_Kiri", out1 => "Data_block_1".data_baru2[8])
   END_RUNG
   RUNG wire#w1
      { S7_Templates := "SrcType := Int" } EQ_Contact(in1 := "Data_block_1".counter_datasuhu, in2 := 10)
      Move(in := "Suhu_Kiri", out1 => "Data_block_1".data_baru2[9])
   END_RUNG
   RUNG wire#w1
      { S7_Templates := "SrcType := Int" } EQ_Contact(in1 := "Data_block_1".counter_datasuhu, in2 := 11)
      Move(in := "Suhu_Kiri", out1 => "Data_block_1".data_baru2[10])
   END_RUNG
   RUNG wire#w1
      { S7_Templates := "SrcType := Int" } EQ_Contact(in1 := "Data_block_1".counter_datasuhu, in2 := 12)
      Move(in := "Suhu_Kiri", out1 => "Data_block_1".data_baru2[11])
   END_RUNG
   RUNG wire#w1
      { S7_Templates := "SrcType := Int" } EQ_Contact(in1 := "Data_block_1".counter_datasuhu, in2 := 13)
      Move(in := "Suhu_Kiri", out1 => "Data_block_1".data_baru2[12])
   END_RUNG
   RUNG wire#w1
      { S7_Templates := "SrcType := Int" } EQ_Contact(in1 := "Data_block_1".counter_datasuhu, in2 := 14)
      Move(in := "Suhu_Kiri", out1 => "Data_block_1".data_baru2[13])
   END_RUNG
   RUNG wire#w1
      { S7_Templates := "SrcType := Int" } EQ_Contact(in1 := "Data_block_1".counter_datasuhu, in2 := 15)
      Move(in := "Suhu_Kiri", out1 => "Data_block_1".data_baru2[14])
   END_RUNG
   RUNG wire#w1
      { S7_Templates := "SrcType := Int" } EQ_Contact(in1 := "Data_block_1".counter_datasuhu, in2 := 16)
      Move(in := "Suhu_Kiri", out1 => "Data_block_1".data_baru2[15])
   END_RUNG
   RUNG wire#w1
      { S7_Templates := "SrcType := Int" } EQ_Contact(in1 := "Data_block_1".counter_datasuhu, in2 := 17)
      Move(in := "Suhu_Kiri", out1 => "Data_block_1".data_baru2[16])
   END_RUNG
   RUNG wire#w1
      { S7_Templates := "SrcType := Int" } EQ_Contact(in1 := "Data_block_1".counter_datasuhu, in2 := 18)
      Move(in := "Suhu_Kiri", out1 => "Data_block_1".data_baru2[17])
   END_RUNG
   RUNG wire#w1
      { S7_Templates := "SrcType := Int" } EQ_Contact(in1 := "Data_block_1".counter_datasuhu, in2 := 19)
      Move(in := "Suhu_Kiri", out1 => "Data_block_1".data_baru2[18])
   END_RUNG
   RUNG wire#w1
      { S7_Templates := "SrcType := Int" } EQ_Contact(in1 := "Data_block_1".counter_datasuhu, in2 := 20)
      Move(in := "Suhu_Kiri", out1 => "Data_block_1".data_baru2[19])
   END_RUNG
   RUNG wire#w1
      { S7_Templates := "SrcType := Int" } EQ_Contact(in1 := "Data_block_1".counter_datasuhu, in2 := 21)
      Move(in := "Suhu_Kiri", out1 => "Data_block_1".data_baru2[20])
   END_RUNG
   RUNG wire#w1
      { S7_Templates := "SrcType := Int" } EQ_Contact(in1 := "Data_block_1".counter_datasuhu, in2 := 22)
      Move(in := "Suhu_Kiri", out1 => "Data_block_1".data_baru2[21])
   END_RUNG
   RUNG wire#w1
      { S7_Templates := "SrcType := Int" } EQ_Contact(in1 := "Data_block_1".counter_datasuhu, in2 := 23)
      Move(in := "Suhu_Kiri", out1 => "Data_block_1".data_baru2[22])
   END_RUNG
   RUNG wire#w1
      { S7_Templates := "SrcType := Int" } EQ_Contact(in1 := "Data_block_1".counter_datasuhu, in2 := 24)
      Move(in := "Suhu_Kiri", out1 => "Data_block_1".data_baru2[23])
   END_RUNG
   RUNG wire#w1
      { S7_Templates := "SrcType := Int" } EQ_Contact(in1 := "Data_block_1".counter_datasuhu, in2 := 25)
      Move(in := "Suhu_Kiri", out1 => "Data_block_1".data_baru2[24])
   END_RUNG
   RUNG wire#w1
      { S7_Templates := "SrcType := Int" } EQ_Contact(in1 := "Data_block_1".counter_datasuhu, in2 := 26)
      Move(in := "Suhu_Kiri", out1 => "Data_block_1".data_baru2[25])
   END_RUNG
   RUNG wire#w1
      { S7_Templates := "SrcType := Int" } EQ_Contact(in1 := "Data_block_1".counter_datasuhu, in2 := 27)
      Move(in := "Suhu_Kiri", out1 => "Data_block_1".data_baru2[26])
   END_RUNG
   RUNG wire#w1
      { S7_Templates := "SrcType := Int" } EQ_Contact(in1 := "Data_block_1".counter_datasuhu, in2 := 28)
      Move(in := "Suhu_Kiri", out1 => "Data_block_1".data_baru2[27])
   END_RUNG
   RUNG wire#w1
      { S7_Templates := "SrcType := Int" } EQ_Contact(in1 := "Data_block_1".counter_datasuhu, in2 := 29)
      Move(in := "Suhu_Kiri", out1 => "Data_block_1".data_baru2[28])
   END_RUNG
   RUNG wire#w1
      { S7_Templates := "SrcType := Int" } EQ_Contact(in1 := "Data_block_1".counter_datasuhu, in2 := 30)
      Move(in := "Suhu_Kiri", out1 => "Data_block_1".data_baru2[29])
   END_RUNG
   RUNG wire#w1
      { S7_Templates := "SrcType := Int" } EQ_Contact(in1 := "Data_block_1".counter_datasuhu, in2 := 31)
      Move(in := "Suhu_Kiri", out1 => "Data_block_1".data_baru2[30])
   END_RUNG
   RUNG wire#w1
      { S7_Templates := "SrcType := Int" } EQ_Contact(in1 := "Data_block_1".counter_datasuhu, in2 := 32)
      Move(in := "Suhu_Kiri", out1 => "Data_block_1".data_baru2[31])
   END_RUNG
   RUNG wire#w1
      { S7_Templates := "SrcType := Int" } EQ_Contact(in1 := "Data_block_1".counter_datasuhu, in2 := 33)
      Move(in := "Suhu_Kiri", out1 => "Data_block_1".data_baru2[32])
   END_RUNG
   RUNG wire#w1
      { S7_Templates := "SrcType := Int" } EQ_Contact(in1 := "Data_block_1".counter_datasuhu, in2 := 34)
      Move(in := "Suhu_Kiri", out1 => "Data_block_1".data_baru2[33])
   END_RUNG
   RUNG wire#w1
      { S7_Templates := "SrcType := Int" } EQ_Contact(in1 := "Data_block_1".counter_datasuhu, in2 := 35)
      Move(in := "Suhu_Kiri", out1 => "Data_block_1".data_baru2[34])
   END_RUNG
   RUNG wire#w1
      { S7_Templates := "SrcType := Int" } EQ_Contact(in1 := "Data_block_1".counter_datasuhu, in2 := 36)
      Move(in := "Suhu_Kiri", out1 => "Data_block_1".data_baru2[35])
   END_RUNG
   RUNG wire#w1
      { S7_Templates := "SrcType := Int" } EQ_Contact(in1 := "Data_block_1".counter_datasuhu, in2 := 37)
      Move(in := "Suhu_Kiri", out1 => "Data_block_1".data_baru2[36])
   END_RUNG
   RUNG wire#w1
      { S7_Templates := "SrcType := Int" } EQ_Contact(in1 := "Data_block_1".counter_datasuhu, in2 := 38)
      Move(in := "Suhu_Kiri", out1 => "Data_block_1".data_baru2[37])
   END_RUNG
   RUNG wire#w1
      { S7_Templates := "SrcType := Int" } EQ_Contact(in1 := "Data_block_1".counter_datasuhu, in2 := 39)
      Move(in := "Suhu_Kiri", out1 => "Data_block_1".data_baru2[38])
   END_RUNG
   RUNG wire#w1
      { S7_Templates := "SrcType := Int" } EQ_Contact(in1 := "Data_block_1".counter_datasuhu, in2 := 40)
      Move(in := "Suhu_Kiri", out1 => "Data_block_1".data_baru2[39])
   END_RUNG
   RUNG wire#w1
      { S7_Templates := "SrcType := Int" } EQ_Contact(in1 := "Data_block_1".counter_datasuhu, in2 := 41)
      Move(in := "Suhu_Kiri", out1 => "Data_block_1".data_baru2[40])
   END_RUNG
   RUNG wire#w1
      { S7_Templates := "SrcType := Int" } EQ_Contact(in1 := "Data_block_1".counter_datasuhu, in2 := 42)
      Move(in := "Suhu_Kiri", out1 => "Data_block_1".data_baru2[41])
   END_RUNG
   RUNG wire#w1
      { S7_Templates := "SrcType := Int" } EQ_Contact(in1 := "Data_block_1".counter_datasuhu, in2 := 43)
      Move(in := "Suhu_Kiri", out1 => "Data_block_1".data_baru2[42])
   END_RUNG
   RUNG wire#w1
      { S7_Templates := "SrcType := Int" } EQ_Contact(in1 := "Data_block_1".counter_datasuhu, in2 := 44)
      Move(in := "Suhu_Kiri", out1 => "Data_block_1".data_baru2[43])
   END_RUNG
   RUNG wire#w1
      { S7_Templates := "SrcType := Int" } EQ_Contact(in1 := "Data_block_1".counter_datasuhu, in2 := 45)
      Move(in := "Suhu_Kiri", out1 => "Data_block_1".data_baru2[44])
   END_RUNG
   RUNG wire#w1
      { S7_Templates := "SrcType := Int" } EQ_Contact(in1 := "Data_block_1".counter_datasuhu, in2 := 46)
      Move(in := "Suhu_Kiri", out1 => "Data_block_1".data_baru2[45])
   END_RUNG
   RUNG wire#w1
      { S7_Templates := "SrcType := Int" } EQ_Contact(in1 := "Data_block_1".counter_datasuhu, in2 := 47)
      Move(in := "Suhu_Kiri", out1 => "Data_block_1".data_baru2[46])
   END_RUNG
   RUNG wire#w1
      { S7_Templates := "SrcType := Int" } EQ_Contact(in1 := "Data_block_1".counter_datasuhu, in2 := 48)
      Move(in := "Suhu_Kiri", out1 => "Data_block_1".data_baru2[47])
   END_RUNG
   RUNG wire#w1
      { S7_Templates := "SrcType := Int" } EQ_Contact(in1 := "Data_block_1".counter_datasuhu, in2 := 49)
      Move(in := "Suhu_Kiri", out1 => "Data_block_1".data_baru2[48])
   END_RUNG
   RUNG wire#w1
      { S7_Templates := "SrcType := Int" } EQ_Contact(in1 := "Data_block_1".counter_datasuhu, in2 := 50)
      Move(in := "Suhu_Kiri", out1 => "Data_block_1".data_baru2[49])
   END_RUNG
   RUNG wire#w1
      { S7_Templates := "SrcType := Int" } EQ_Contact(in1 := "Data_block_1".counter_datasuhu, in2 := 51)
      Move(in := "Suhu_Kiri", out1 => "Data_block_1".data_baru2[50])
   END_RUNG
   RUNG wire#w1
      { S7_Templates := "SrcType := Int" } EQ_Contact(in1 := "Data_block_1".counter_datasuhu, in2 := 52)
      Move(in := "Suhu_Kiri", out1 => "Data_block_1".data_baru2[51])
   END_RUNG
   RUNG wire#w1
      { S7_Templates := "SrcType := Int" } EQ_Contact(in1 := "Data_block_1".counter_datasuhu, in2 := 53)
      Move(in := "Suhu_Kiri", out1 => "Data_block_1".data_baru2[52])
   END_RUNG
   RUNG wire#w1
      { S7_Templates := "SrcType := Int" } EQ_Contact(in1 := "Data_block_1".counter_datasuhu, in2 := 54)
      Move(in := "Suhu_Kiri", out1 => "Data_block_1".data_baru2[53])
   END_RUNG
   RUNG wire#w1
      { S7_Templates := "SrcType := Int" } EQ_Contact(in1 := "Data_block_1".counter_datasuhu, in2 := 55)
      Move(in := "Suhu_Kiri", out1 => "Data_block_1".data_baru2[54])
   END_RUNG
   RUNG wire#w1
      { S7_Templates := "SrcType := Int" } EQ_Contact(in1 := "Data_block_1".counter_datasuhu, in2 := 56)
      Move(in := "Suhu_Kiri", out1 => "Data_block_1".data_baru2[55])
   END_RUNG
   RUNG wire#w1
      { S7_Templates := "SrcType := Int" } EQ_Contact(in1 := "Data_block_1".counter_datasuhu, in2 := 57)
      Move(in := "Suhu_Kiri", out1 => "Data_block_1".data_baru2[56])
   END_RUNG
   RUNG wire#w1
      { S7_Templates := "SrcType := Int" } EQ_Contact(in1 := "Data_block_1".counter_datasuhu, in2 := 58)
      Move(in := "Suhu_Kiri", out1 => "Data_block_1".data_baru2[57])
   END_RUNG
   RUNG wire#w1
      { S7_Templates := "SrcType := Int" } EQ_Contact(in1 := "Data_block_1".counter_datasuhu, in2 := 59)
      Move(in := "Suhu_Kiri", out1 => "Data_block_1".data_baru2[58])
   END_RUNG
   RUNG wire#w1
      { S7_Templates := "SrcType := Int" } EQ_Contact(in1 := "Data_block_1".counter_datasuhu, in2 := 60)
      Move(in := "Suhu_Kiri", out1 => "Data_block_1".data_baru2[59])
   END_RUNG
   RUNG wire#w1
      { S7_Templates := "SrcType := Int" } EQ_Contact(in1 := "Data_block_1".counter_datasuhu, in2 := 61)
      Move(in := "Suhu_Kiri", out1 => "Data_block_1".data_baru2[60])
   END_RUNG
   RUNG wire#w1
      { S7_Templates := "SrcType := Int" } EQ_Contact(in1 := "Data_block_1".counter_datasuhu, in2 := 62)
      Move(in := "Suhu_Kiri", out1 => "Data_block_1".data_baru2[61])
   END_RUNG
   RUNG wire#w1
      { S7_Templates := "SrcType := Int" } EQ_Contact(in1 := "Data_block_1".counter_datasuhu, in2 := 63)
      Move(in := "Suhu_Kiri", out1 => "Data_block_1".data_baru2[62])
   END_RUNG
   RUNG wire#w1
      { S7_Templates := "SrcType := Int" } EQ_Contact(in1 := "Data_block_1".counter_datasuhu, in2 := 64)
      Move(in := "Suhu_Kiri", out1 => "Data_block_1".data_baru2[63])
   END_RUNG
   RUNG wire#w1
      { S7_Templates := "SrcType := Int" } EQ_Contact(in1 := "Data_block_1".counter_datasuhu, in2 := 65)
      Move(in := "Suhu_Kiri", out1 => "Data_block_1".data_baru2[64])
   END_RUNG
   RUNG wire#w1
      { S7_Templates := "SrcType := Int" } EQ_Contact(in1 := "Data_block_1".counter_datasuhu, in2 := 66)
      Move(in := "Suhu_Kiri", out1 => "Data_block_1".data_baru2[65])
   END_RUNG
   RUNG wire#w1
      { S7_Templates := "SrcType := Int" } EQ_Contact(in1 := "Data_block_1".counter_datasuhu, in2 := 67)
      Move(in := "Suhu_Kiri", out1 => "Data_block_1".data_baru2[66])
   END_RUNG
   RUNG wire#w1
      { S7_Templates := "SrcType := Int" } EQ_Contact(in1 := "Data_block_1".counter_datasuhu, in2 := 68)
      Move(in := "Suhu_Kiri", out1 => "Data_block_1".data_baru2[67])
   END_RUNG
   RUNG wire#w1
      { S7_Templates := "SrcType := Int" } EQ_Contact(in1 := "Data_block_1".counter_datasuhu, in2 := 69)
      Move(in := "Suhu_Kiri", out1 => "Data_block_1".data_baru2[68])
   END_RUNG
   RUNG wire#w1
      { S7_Templates := "SrcType := Int" } EQ_Contact(in1 := "Data_block_1".counter_datasuhu, in2 := 70)
      Move(in := "Suhu_Kiri", out1 => "Data_block_1".data_baru2[69])
   END_RUNG
   RUNG wire#w1
      { S7_Templates := "SrcType := Int" } EQ_Contact(in1 := "Data_block_1".counter_datasuhu, in2 := 71)
      Move(in := "Suhu_Kiri", out1 => "Data_block_1".data_baru2[70])
   END_RUNG
   RUNG wire#w1
      { S7_Templates := "SrcType := Int" } EQ_Contact(in1 := "Data_block_1".counter_datasuhu, in2 := 72)
      Move(in := "Suhu_Kiri", out1 => "Data_block_1".data_baru2[71])
   END_RUNG
   RUNG wire#w1
      { S7_Templates := "SrcType := Int" } EQ_Contact(in1 := "Data_block_1".counter_datasuhu, in2 := 73)
      Move(in := "Suhu_Kiri", out1 => "Data_block_1".data_baru2[72])
   END_RUNG
   RUNG wire#w1
      { S7_Templates := "SrcType := Int" } EQ_Contact(in1 := "Data_block_1".counter_datasuhu, in2 := 74)
      Move(in := "Suhu_Kiri", out1 => "Data_block_1".data_baru2[73])
   END_RUNG
   RUNG wire#w1
      { S7_Templates := "SrcType := Int" } EQ_Contact(in1 := "Data_block_1".counter_datasuhu, in2 := 75)
      Move(in := "Suhu_Kiri", out1 => "Data_block_1".data_baru2[74])
   END_RUNG
   RUNG wire#w1
      { S7_Templates := "SrcType := Int" } EQ_Contact(in1 := "Data_block_1".counter_datasuhu, in2 := 76)
      Move(in := "Suhu_Kiri", out1 => "Data_block_1".data_baru2[75])
   END_RUNG
   RUNG wire#w1
      { S7_Templates := "SrcType := Int" } EQ_Contact(in1 := "Data_block_1".counter_datasuhu, in2 := 77)
      Move(in := "Suhu_Kiri", out1 => "Data_block_1".data_baru2[76])
   END_RUNG
   RUNG wire#w1
      { S7_Templates := "SrcType := Int" } EQ_Contact(in1 := "Data_block_1".counter_datasuhu, in2 := 78)
      Move(in := "Suhu_Kiri", out1 => "Data_block_1".data_baru2[77])
   END_RUNG
   RUNG wire#w1
      { S7_Templates := "SrcType := Int" } EQ_Contact(in1 := "Data_block_1".counter_datasuhu, in2 := 79)
      Move(in := "Suhu_Kiri", out1 => "Data_block_1".data_baru2[78])
   END_RUNG
   RUNG wire#w1
      { S7_Templates := "SrcType := Int" } EQ_Contact(in1 := "Data_block_1".counter_datasuhu, in2 := 80)
      Move(in := "Suhu_Kiri", out1 => "Data_block_1".data_baru2[79])
   END_RUNG
   RUNG wire#w1
      { S7_Templates := "SrcType := Int" } EQ_Contact(in1 := "Data_block_1".counter_datasuhu, in2 := 81)
      Move(in := "Suhu_Kiri", out1 => "Data_block_1".data_baru2[80])
   END_RUNG
   RUNG wire#w1
      { S7_Templates := "SrcType := Int" } EQ_Contact(in1 := "Data_block_1".counter_datasuhu, in2 := 82)
      Move(in := "Suhu_Kiri", out1 => "Data_block_1".data_baru2[81])
   END_RUNG
   RUNG wire#w1
      { S7_Templates := "SrcType := Int" } EQ_Contact(in1 := "Data_block_1".counter_datasuhu, in2 := 83)
      Move(in := "Suhu_Kiri", out1 => "Data_block_1".data_baru2[82])
   END_RUNG
   RUNG wire#w1
      { S7_Templates := "SrcType := Int" } EQ_Contact(in1 := "Data_block_1".counter_datasuhu, in2 := 84)
      Move(in := "Suhu_Kiri", out1 => "Data_block_1".data_baru2[83])
   END_RUNG
   RUNG wire#w1
      { S7_Templates := "SrcType := Int" } EQ_Contact(in1 := "Data_block_1".counter_datasuhu, in2 := 85)
      Move(in := "Suhu_Kiri", out1 => "Data_block_1".data_baru2[84])
   END_RUNG
   RUNG wire#w1
      { S7_Templates := "SrcType := Int" } EQ_Contact(in1 := "Data_block_1".counter_datasuhu, in2 := 86)
      Move(in := "Suhu_Kiri", out1 => "Data_block_1".data_baru2[85])
   END_RUNG
   RUNG wire#w1
      { S7_Templates := "SrcType := Int" } EQ_Contact(in1 := "Data_block_1".counter_datasuhu, in2 := 87)
      Move(in := "Suhu_Kiri", out1 => "Data_block_1".data_baru2[86])
   END_RUNG
   RUNG wire#w1
      { S7_Templates := "SrcType := Int" } EQ_Contact(in1 := "Data_block_1".counter_datasuhu, in2 := 88)
      Move(in := "Suhu_Kiri", out1 => "Data_block_1".data_baru2[87])
   END_RUNG
   RUNG wire#w1
      { S7_Templates := "SrcType := Int" } EQ_Contact(in1 := "Data_block_1".counter_datasuhu, in2 := 89)
      Move(in := "Suhu_Kiri", out1 => "Data_block_1".data_baru2[88])
   END_RUNG
   RUNG wire#w1
      { S7_Templates := "SrcType := Int" } EQ_Contact(in1 := "Data_block_1".counter_datasuhu, in2 := 90)
      Move(in := "Suhu_Kiri", out1 => "Data_block_1".data_baru2[89])
   END_RUNG
   RUNG wire#w1
      { S7_Templates := "SrcType := Int" } EQ_Contact(in1 := "Data_block_1".counter_datasuhu, in2 := 91)
      Move(in := "Suhu_Kiri", out1 => "Data_block_1".data_baru2[90])
   END_RUNG
   RUNG wire#w1
      { S7_Templates := "SrcType := Int" } EQ_Contact(in1 := "Data_block_1".counter_datasuhu, in2 := 92)
      Move(in := "Suhu_Kiri", out1 => "Data_block_1".data_baru2[91])
   END_RUNG
   RUNG wire#w1
      { S7_Templates := "SrcType := Int" } EQ_Contact(in1 := "Data_block_1".counter_datasuhu, in2 := 93)
      Move(in := "Suhu_Kiri", out1 => "Data_block_1".data_baru2[92])
   END_RUNG
   RUNG wire#w1
      { S7_Templates := "SrcType := Int" } EQ_Contact(in1 := "Data_block_1".counter_datasuhu, in2 := 94)
      Move(in := "Suhu_Kiri", out1 => "Data_block_1".data_baru2[93])
   END_RUNG
   RUNG wire#w1
      { S7_Templates := "SrcType := Int" } EQ_Contact(in1 := "Data_block_1".counter_datasuhu, in2 := 95)
      Move(in := "Suhu_Kiri", out1 => "Data_block_1".data_baru2[94])
   END_RUNG
   RUNG wire#w1
      { S7_Templates := "SrcType := Int" } EQ_Contact(in1 := "Data_block_1".counter_datasuhu, in2 := 96)
      Move(in := "Suhu_Kiri", out1 => "Data_block_1".data_baru2[95])
   END_RUNG
   RUNG wire#w1
      { S7_Templates := "SrcType := Int" } EQ_Contact(in1 := "Data_block_1".counter_datasuhu, in2 := 97)
      Move(in := "Suhu_Kiri", out1 => "Data_block_1".data_baru2[96])
   END_RUNG
   RUNG wire#w1
      { S7_Templates := "SrcType := Int" } EQ_Contact(in1 := "Data_block_1".counter_datasuhu, in2 := 98)
      Move(in := "Suhu_Kiri", out1 => "Data_block_1".data_baru2[97])
   END_RUNG
   RUNG wire#w1
      { S7_Templates := "SrcType := Int" } EQ_Contact(in1 := "Data_block_1".counter_datasuhu, in2 := 99)
      Move(in := "Suhu_Kiri", out1 => "Data_block_1".data_baru2[98])
   END_RUNG
   RUNG wire#w1
      { S7_Templates := "SrcType := Int" } EQ_Contact(in1 := "Data_block_1".counter_datasuhu, in2 := 100)
      Move(in := "Suhu_Kiri", out1 => "Data_block_1".data_baru2[99])
   END_RUNG
   // the same network as SCL:
   #_w1 := "Data_block_1".K2 AND NOT "Data_block_1".Lock_A;
   IF #_w1 AND ("Data_block_1".counter_datasuhu = 1) THEN
       "Data_block_1".data_baru2[0] := "Suhu_Kiri";
   END_IF;
   IF #_w1 AND ("Data_block_1".counter_datasuhu = 2) THEN
       "Data_block_1".data_baru2[1] := "Suhu_Kiri";
   END_IF;
   IF #_w1 AND ("Data_block_1".counter_datasuhu = 3) THEN
       "Data_block_1".data_baru2[2] := "Suhu_Kiri";
   END_IF;
   IF #_w1 AND ("Data_block_1".counter_datasuhu = 4) THEN
       "Data_block_1".data_baru2[3] := "Suhu_Kiri";
   END_IF;
   IF #_w1 AND ("Data_block_1".counter_datasuhu = 5) THEN
       "Data_block_1".data_baru2[4] := "Suhu_Kiri";
   END_IF;
   IF #_w1 AND ("Data_block_1".counter_datasuhu = 6) THEN
       "Data_block_1".data_baru2[5] := "Suhu_Kiri";
   END_IF;
   IF #_w1 AND ("Data_block_1".counter_datasuhu = 7) THEN
       "Data_block_1".data_baru2[6] := "Suhu_Kiri";
   END_IF;
   IF #_w1 AND ("Data_block_1".counter_datasuhu = 8) THEN
       "Data_block_1".data_baru2[7] := "Suhu_Kiri";
   END_IF;
   IF #_w1 AND ("Data_block_1".counter_datasuhu = 9) THEN
       "Data_block_1".data_baru2[8] := "Suhu_Kiri";
   END_IF;
   IF #_w1 AND ("Data_block_1".counter_datasuhu = 10) THEN
       "Data_block_1".data_baru2[9] := "Suhu_Kiri";
   END_IF;
   IF #_w1 AND ("Data_block_1".counter_datasuhu = 11) THEN
       "Data_block_1".data_baru2[10] := "Suhu_Kiri";
   END_IF;
   IF #_w1 AND ("Data_block_1".counter_datasuhu = 12) THEN
       "Data_block_1".data_baru2[11] := "Suhu_Kiri";
   END_IF;
   IF #_w1 AND ("Data_block_1".counter_datasuhu = 13) THEN
       "Data_block_1".data_baru2[12] := "Suhu_Kiri";
   END_IF;
   IF #_w1 AND ("Data_block_1".counter_datasuhu = 14) THEN
       "Data_block_1".data_baru2[13] := "Suhu_Kiri";
   END_IF;
   IF #_w1 AND ("Data_block_1".counter_datasuhu = 15) THEN
       "Data_block_1".data_baru2[14] := "Suhu_Kiri";
   END_IF;
   IF #_w1 AND ("Data_block_1".counter_datasuhu = 16) THEN
       "Data_block_1".data_baru2[15] := "Suhu_Kiri";
   END_IF;
   IF #_w1 AND ("Data_block_1".counter_datasuhu = 17) THEN
       "Data_block_1".data_baru2[16] := "Suhu_Kiri";
   END_IF;
   IF #_w1 AND ("Data_block_1".counter_datasuhu = 18) THEN
       "Data_block_1".data_baru2[17] := "Suhu_Kiri";
   END_IF;
   IF #_w1 AND ("Data_block_1".counter_datasuhu = 19) THEN
       "Data_block_1".data_baru2[18] := "Suhu_Kiri";
   END_IF;
   IF #_w1 AND ("Data_block_1".counter_datasuhu = 20) THEN
       "Data_block_1".data_baru2[19] := "Suhu_Kiri";
   END_IF;
   IF #_w1 AND ("Data_block_1".counter_datasuhu = 21) THEN
       "Data_block_1".data_baru2[20] := "Suhu_Kiri";
   END_IF;
   IF #_w1 AND ("Data_block_1".counter_datasuhu = 22) THEN
       "Data_block_1".data_baru2[21] := "Suhu_Kiri";
   END_IF;
   IF #_w1 AND ("Data_block_1".counter_datasuhu = 23) THEN
       "Data_block_1".data_baru2[22] := "Suhu_Kiri";
   END_IF;
   IF #_w1 AND ("Data_block_1".counter_datasuhu = 24) THEN
       "Data_block_1".data_baru2[23] := "Suhu_Kiri";
   END_IF;
   IF #_w1 AND ("Data_block_1".counter_datasuhu = 25) THEN
       "Data_block_1".data_baru2[24] := "Suhu_Kiri";
   END_IF;
   IF #_w1 AND ("Data_block_1".counter_datasuhu = 26) THEN
       "Data_block_1".data_baru2[25] := "Suhu_Kiri";
   END_IF;
   IF #_w1 AND ("Data_block_1".counter_datasuhu = 27) THEN
       "Data_block_1".data_baru2[26] := "Suhu_Kiri";
   END_IF;
   IF #_w1 AND ("Data_block_1".counter_datasuhu = 28) THEN
       "Data_block_1".data_baru2[27] := "Suhu_Kiri";
   END_IF;
   IF #_w1 AND ("Data_block_1".counter_datasuhu = 29) THEN
       "Data_block_1".data_baru2[28] := "Suhu_Kiri";
   END_IF;
   IF #_w1 AND ("Data_block_1".counter_datasuhu = 30) THEN
       "Data_block_1".data_baru2[29] := "Suhu_Kiri";
   END_IF;
   IF #_w1 AND ("Data_block_1".counter_datasuhu = 31) THEN
       "Data_block_1".data_baru2[30] := "Suhu_Kiri";
   END_IF;
   IF #_w1 AND ("Data_block_1".counter_datasuhu = 32) THEN
       "Data_block_1".data_baru2[31] := "Suhu_Kiri";
   END_IF;
   IF #_w1 AND ("Data_block_1".counter_datasuhu = 33) THEN
       "Data_block_1".data_baru2[32] := "Suhu_Kiri";
   END_IF;
   IF #_w1 AND ("Data_block_1".counter_datasuhu = 34) THEN
       "Data_block_1".data_baru2[33] := "Suhu_Kiri";
   END_IF;
   IF #_w1 AND ("Data_block_1".counter_datasuhu = 35) THEN
       "Data_block_1".data_baru2[34] := "Suhu_Kiri";
   END_IF;
   IF #_w1 AND ("Data_block_1".counter_datasuhu = 36) THEN
       "Data_block_1".data_baru2[35] := "Suhu_Kiri";
   END_IF;
   IF #_w1 AND ("Data_block_1".counter_datasuhu = 37) THEN
       "Data_block_1".data_baru2[36] := "Suhu_Kiri";
   END_IF;
   IF #_w1 AND ("Data_block_1".counter_datasuhu = 38) THEN
       "Data_block_1".data_baru2[37] := "Suhu_Kiri";
   END_IF;
   IF #_w1 AND ("Data_block_1".counter_datasuhu = 39) THEN
       "Data_block_1".data_baru2[38] := "Suhu_Kiri";
   END_IF;
   IF #_w1 AND ("Data_block_1".counter_datasuhu = 40) THEN
       "Data_block_1".data_baru2[39] := "Suhu_Kiri";
   END_IF;
   IF #_w1 AND ("Data_block_1".counter_datasuhu = 41) THEN
       "Data_block_1".data_baru2[40] := "Suhu_Kiri";
   END_IF;
   IF #_w1 AND ("Data_block_1".counter_datasuhu = 42) THEN
       "Data_block_1".data_baru2[41] := "Suhu_Kiri";
   END_IF;
   IF #_w1 AND ("Data_block_1".counter_datasuhu = 43) THEN
       "Data_block_1".data_baru2[42] := "Suhu_Kiri";
   END_IF;
   IF #_w1 AND ("Data_block_1".counter_datasuhu = 44) THEN
       "Data_block_1".data_baru2[43] := "Suhu_Kiri";
   END_IF;
   IF #_w1 AND ("Data_block_1".counter_datasuhu = 45) THEN
       "Data_block_1".data_baru2[44] := "Suhu_Kiri";
   END_IF;
   IF #_w1 AND ("Data_block_1".counter_datasuhu = 46) THEN
       "Data_block_1".data_baru2[45] := "Suhu_Kiri";
   END_IF;
   IF #_w1 AND ("Data_block_1".counter_datasuhu = 47) THEN
       "Data_block_1".data_baru2[46] := "Suhu_Kiri";
   END_IF;
   IF #_w1 AND ("Data_block_1".counter_datasuhu = 48) THEN
       "Data_block_1".data_baru2[47] := "Suhu_Kiri";
   END_IF;
   IF #_w1 AND ("Data_block_1".counter_datasuhu = 49) THEN
       "Data_block_1".data_baru2[48] := "Suhu_Kiri";
   END_IF;
   IF #_w1 AND ("Data_block_1".counter_datasuhu = 50) THEN
       "Data_block_1".data_baru2[49] := "Suhu_Kiri";
   END_IF;
   IF #_w1 AND ("Data_block_1".counter_datasuhu = 51) THEN
       "Data_block_1".data_baru2[50] := "Suhu_Kiri";
   END_IF;
   IF #_w1 AND ("Data_block_1".counter_datasuhu = 52) THEN
       "Data_block_1".data_baru2[51] := "Suhu_Kiri";
   END_IF;
   IF #_w1 AND ("Data_block_1".counter_datasuhu = 53) THEN
       "Data_block_1".data_baru2[52] := "Suhu_Kiri";
   END_IF;
   IF #_w1 AND ("Data_block_1".counter_datasuhu = 54) THEN
       "Data_block_1".data_baru2[53] := "Suhu_Kiri";
   END_IF;
   IF #_w1 AND ("Data_block_1".counter_datasuhu = 55) THEN
       "Data_block_1".data_baru2[54] := "Suhu_Kiri";
   END_IF;
   IF #_w1 AND ("Data_block_1".counter_datasuhu = 56) THEN
       "Data_block_1".data_baru2[55] := "Suhu_Kiri";
   END_IF;
   IF #_w1 AND ("Data_block_1".counter_datasuhu = 57) THEN
       "Data_block_1".data_baru2[56] := "Suhu_Kiri";
   END_IF;
   IF #_w1 AND ("Data_block_1".counter_datasuhu = 58) THEN
       "Data_block_1".data_baru2[57] := "Suhu_Kiri";
   END_IF;
   IF #_w1 AND ("Data_block_1".counter_datasuhu = 59) THEN
       "Data_block_1".data_baru2[58] := "Suhu_Kiri";
   END_IF;
   IF #_w1 AND ("Data_block_1".counter_datasuhu = 60) THEN
       "Data_block_1".data_baru2[59] := "Suhu_Kiri";
   END_IF;
   IF #_w1 AND ("Data_block_1".counter_datasuhu = 61) THEN
       "Data_block_1".data_baru2[60] := "Suhu_Kiri";
   END_IF;
   IF #_w1 AND ("Data_block_1".counter_datasuhu = 62) THEN
       "Data_block_1".data_baru2[61] := "Suhu_Kiri";
   END_IF;
   IF #_w1 AND ("Data_block_1".counter_datasuhu = 63) THEN
       "Data_block_1".data_baru2[62] := "Suhu_Kiri";
   END_IF;
   IF #_w1 AND ("Data_block_1".counter_datasuhu = 64) THEN
       "Data_block_1".data_baru2[63] := "Suhu_Kiri";
   END_IF;
   IF #_w1 AND ("Data_block_1".counter_datasuhu = 65) THEN
       "Data_block_1".data_baru2[64] := "Suhu_Kiri";
   END_IF;
   IF #_w1 AND ("Data_block_1".counter_datasuhu = 66) THEN
       "Data_block_1".data_baru2[65] := "Suhu_Kiri";
   END_IF;
   IF #_w1 AND ("Data_block_1".counter_datasuhu = 67) THEN
       "Data_block_1".data_baru2[66] := "Suhu_Kiri";
   END_IF;
   IF #_w1 AND ("Data_block_1".counter_datasuhu = 68) THEN
       "Data_block_1".data_baru2[67] := "Suhu_Kiri";
   END_IF;
   IF #_w1 AND ("Data_block_1".counter_datasuhu = 69) THEN
       "Data_block_1".data_baru2[68] := "Suhu_Kiri";
   END_IF;
   IF #_w1 AND ("Data_block_1".counter_datasuhu = 70) THEN
       "Data_block_1".data_baru2[69] := "Suhu_Kiri";
   END_IF;
   IF #_w1 AND ("Data_block_1".counter_datasuhu = 71) THEN
       "Data_block_1".data_baru2[70] := "Suhu_Kiri";
   END_IF;
   IF #_w1 AND ("Data_block_1".counter_datasuhu = 72) THEN
       "Data_block_1".data_baru2[71] := "Suhu_Kiri";
   END_IF;
   IF #_w1 AND ("Data_block_1".counter_datasuhu = 73) THEN
       "Data_block_1".data_baru2[72] := "Suhu_Kiri";
   END_IF;
   IF #_w1 AND ("Data_block_1".counter_datasuhu = 74) THEN
       "Data_block_1".data_baru2[73] := "Suhu_Kiri";
   END_IF;
   IF #_w1 AND ("Data_block_1".counter_datasuhu = 75) THEN
       "Data_block_1".data_baru2[74] := "Suhu_Kiri";
   END_IF;
   IF #_w1 AND ("Data_block_1".counter_datasuhu = 76) THEN
       "Data_block_1".data_baru2[75] := "Suhu_Kiri";
   END_IF;
   IF #_w1 AND ("Data_block_1".counter_datasuhu = 77) THEN
       "Data_block_1".data_baru2[76] := "Suhu_Kiri";
   END_IF;
   IF #_w1 AND ("Data_block_1".counter_datasuhu = 78) THEN
       "Data_block_1".data_baru2[77] := "Suhu_Kiri";
   END_IF;
   IF #_w1 AND ("Data_block_1".counter_datasuhu = 79) THEN
       "Data_block_1".data_baru2[78] := "Suhu_Kiri";
   END_IF;
   IF #_w1 AND ("Data_block_1".counter_datasuhu = 80) THEN
       "Data_block_1".data_baru2[79] := "Suhu_Kiri";
   END_IF;
   IF #_w1 AND ("Data_block_1".counter_datasuhu = 81) THEN
       "Data_block_1".data_baru2[80] := "Suhu_Kiri";
   END_IF;
   IF #_w1 AND ("Data_block_1".counter_datasuhu = 82) THEN
       "Data_block_1".data_baru2[81] := "Suhu_Kiri";
   END_IF;
   IF #_w1 AND ("Data_block_1".counter_datasuhu = 83) THEN
       "Data_block_1".data_baru2[82] := "Suhu_Kiri";
   END_IF;
   IF #_w1 AND ("Data_block_1".counter_datasuhu = 84) THEN
       "Data_block_1".data_baru2[83] := "Suhu_Kiri";
   END_IF;
   IF #_w1 AND ("Data_block_1".counter_datasuhu = 85) THEN
       "Data_block_1".data_baru2[84] := "Suhu_Kiri";
   END_IF;
   IF #_w1 AND ("Data_block_1".counter_datasuhu = 86) THEN
       "Data_block_1".data_baru2[85] := "Suhu_Kiri";
   END_IF;
   IF #_w1 AND ("Data_block_1".counter_datasuhu = 87) THEN
       "Data_block_1".data_baru2[86] := "Suhu_Kiri";
   END_IF;
   IF #_w1 AND ("Data_block_1".counter_datasuhu = 88) THEN
       "Data_block_1".data_baru2[87] := "Suhu_Kiri";
   END_IF;
   IF #_w1 AND ("Data_block_1".counter_datasuhu = 89) THEN
       "Data_block_1".data_baru2[88] := "Suhu_Kiri";
   END_IF;
   IF #_w1 AND ("Data_block_1".counter_datasuhu = 90) THEN
       "Data_block_1".data_baru2[89] := "Suhu_Kiri";
   END_IF;
   IF #_w1 AND ("Data_block_1".counter_datasuhu = 91) THEN
       "Data_block_1".data_baru2[90] := "Suhu_Kiri";
   END_IF;
   IF #_w1 AND ("Data_block_1".counter_datasuhu = 92) THEN
       "Data_block_1".data_baru2[91] := "Suhu_Kiri";
   END_IF;
   IF #_w1 AND ("Data_block_1".counter_datasuhu = 93) THEN
       "Data_block_1".data_baru2[92] := "Suhu_Kiri";
   END_IF;
   IF #_w1 AND ("Data_block_1".counter_datasuhu = 94) THEN
       "Data_block_1".data_baru2[93] := "Suhu_Kiri";
   END_IF;
   IF #_w1 AND ("Data_block_1".counter_datasuhu = 95) THEN
       "Data_block_1".data_baru2[94] := "Suhu_Kiri";
   END_IF;
   IF #_w1 AND ("Data_block_1".counter_datasuhu = 96) THEN
       "Data_block_1".data_baru2[95] := "Suhu_Kiri";
   END_IF;
   IF #_w1 AND ("Data_block_1".counter_datasuhu = 97) THEN
       "Data_block_1".data_baru2[96] := "Suhu_Kiri";
   END_IF;
   IF #_w1 AND ("Data_block_1".counter_datasuhu = 98) THEN
       "Data_block_1".data_baru2[97] := "Suhu_Kiri";
   END_IF;
   IF #_w1 AND ("Data_block_1".counter_datasuhu = 99) THEN
       "Data_block_1".data_baru2[98] := "Suhu_Kiri";
   END_IF;
   IF #_w1 AND ("Data_block_1".counter_datasuhu = 100) THEN
       "Data_block_1".data_baru2[99] := "Suhu_Kiri";
   END_IF;
END_REGION

REGION Network 11: Mengolah Data (kanan ke kiri)
   // program ketika sensor prox b tidak aktif, maka akan mengaktifkan pemutus, menambah counter, mengubah roda ke- (angka genap dari 2-38) (sisi kanan) (angka ganjil dari 1-37) (sisi kiri)
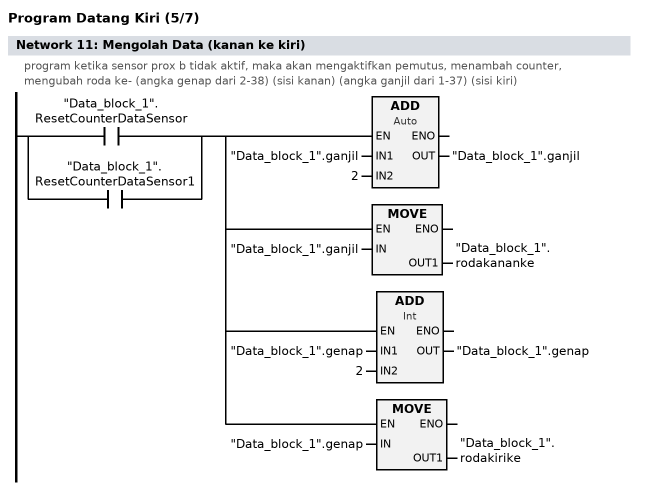
   RUNG wire#powerrail
      Contact( "Data_block_1".ResetCounterDataSensor )
      wire#w1
      Add(in1 := "Data_block_1".ganjil, in2 := 2, out => "Data_block_1".ganjil)
   END_RUNG
   RUNG wire#powerrail
      Contact( "Data_block_1".ResetCounterDataSensor1 )
   END_RUNG wire#w1
   RUNG wire#w1
      Move(in := "Data_block_1".ganjil, out1 => "Data_block_1".rodakananke)
   END_RUNG
   RUNG wire#w1
      { S7_Templates := "SrcType := Int" } Add(in1 := "Data_block_1".genap, in2 := 2, out => "Data_block_1".genap)
   END_RUNG
   RUNG wire#w1
      Move(in := "Data_block_1".genap, out1 => "Data_block_1".rodakirike)
   END_RUNG
   // the same network as SCL:
   IF "Data_block_1".ResetCounterDataSensor OR "Data_block_1".ResetCounterDataSensor1 THEN
       "Data_block_1".ganjil := "Data_block_1".ganjil + 2;
       "Data_block_1".rodakananke := "Data_block_1".ganjil;
       "Data_block_1".genap := "Data_block_1".genap + 2;
       "Data_block_1".rodakirike := "Data_block_1".genap;
   END_IF;
END_REGION

REGION Network 12: Memasukkan Data
   // ketika pemutus aktif dan counter bertambah, data suhu lama dipindahkan ke array dataroda (dari 0-37) serta sarana akan ditampilkan pada tabel sesuai roda pertama tiap sarana
   // ketika pemutus aktif, data suhu, data suhu lama , dan data suhu baru akan menjadi 0
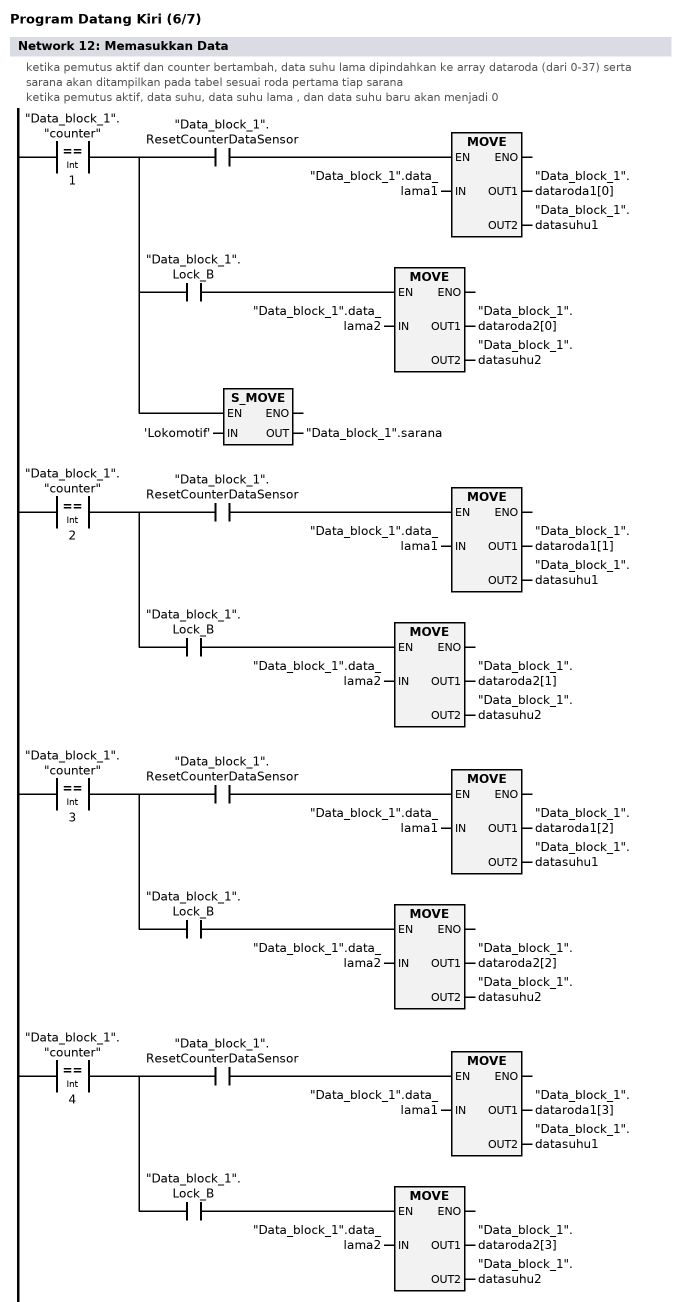
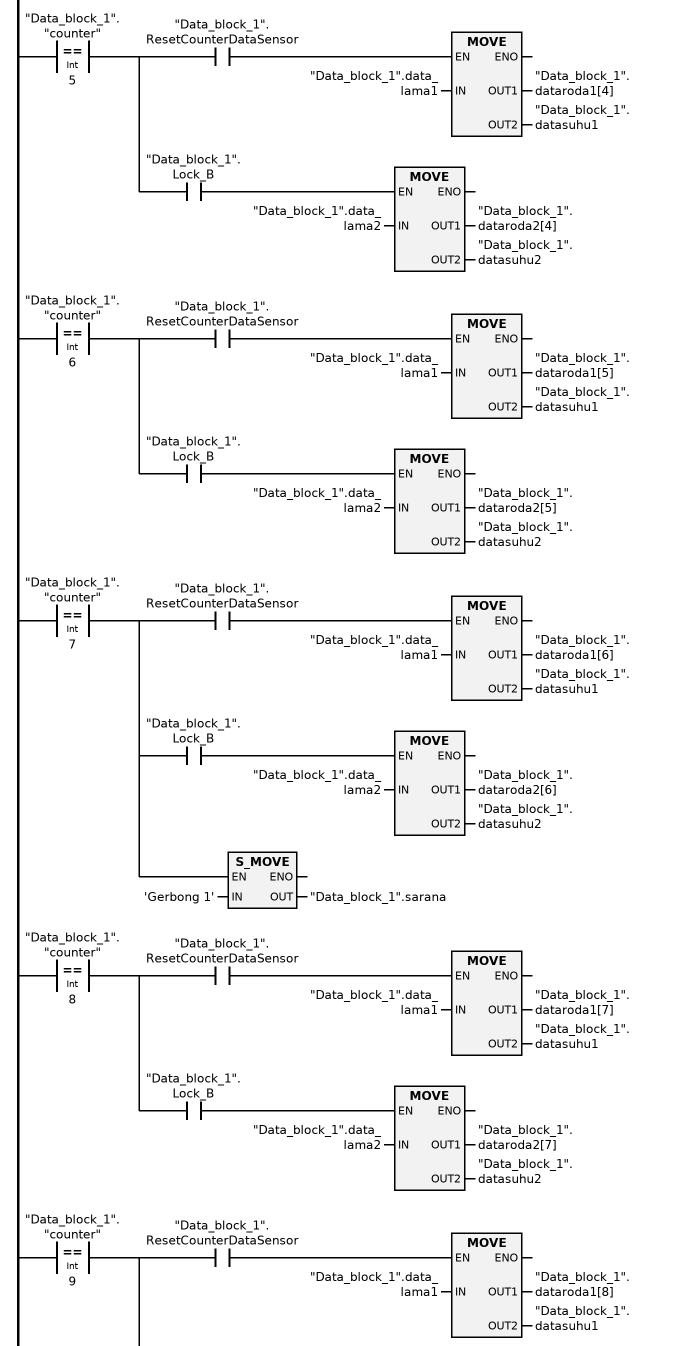
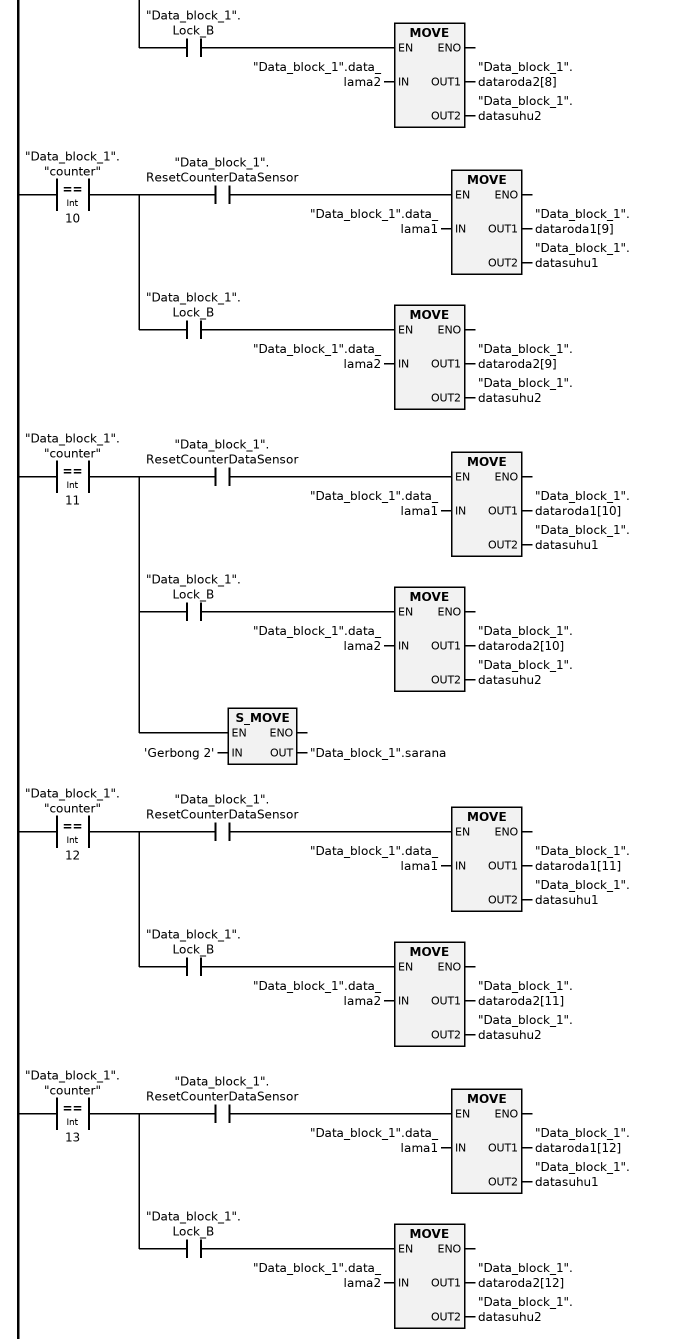
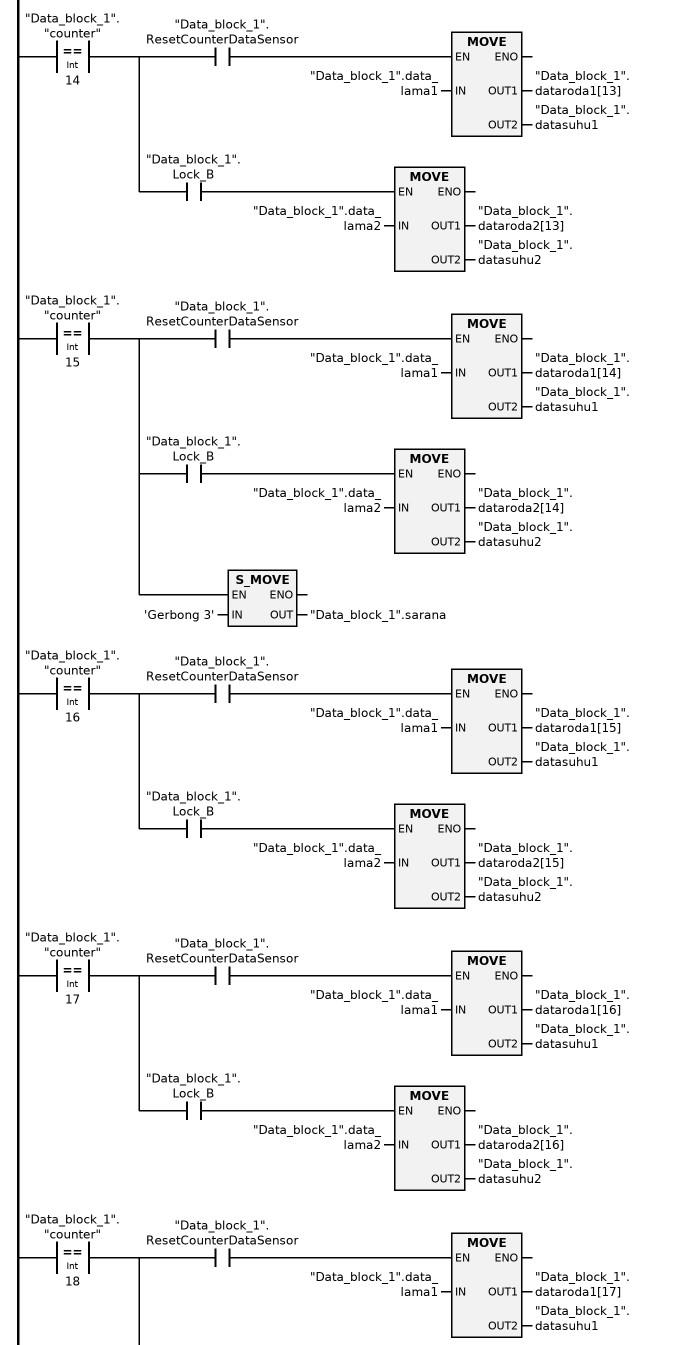
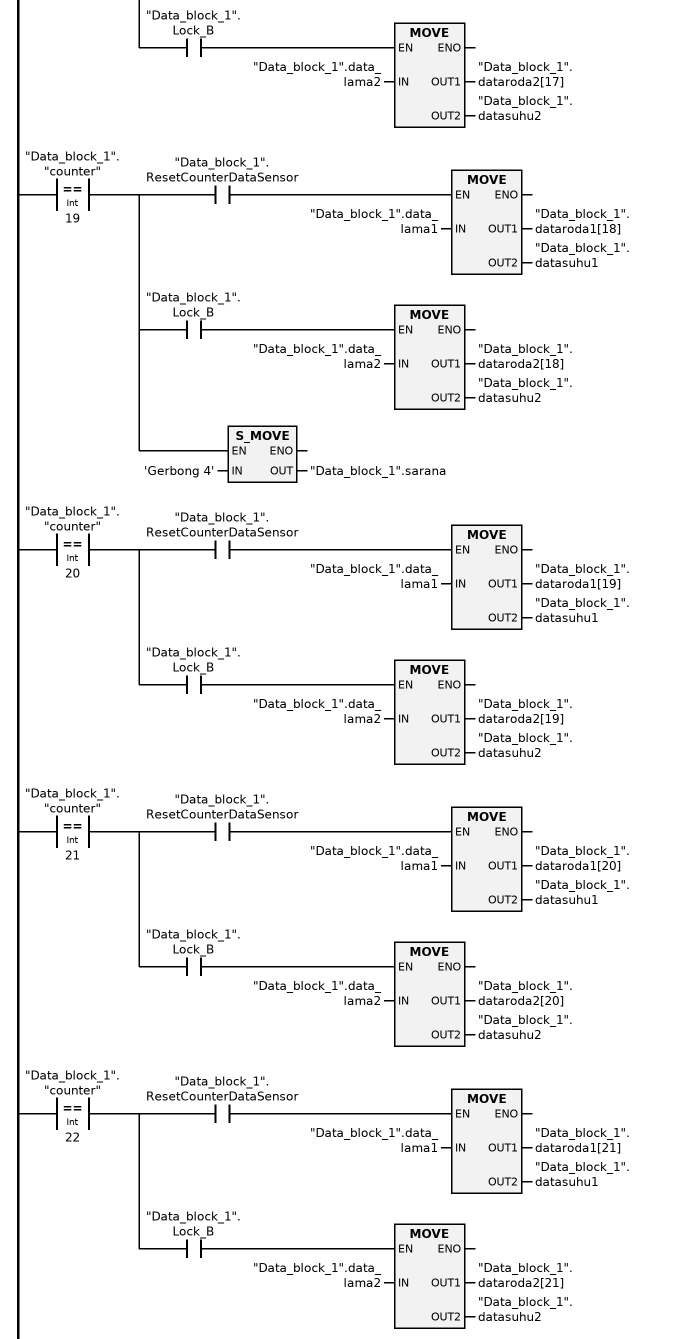
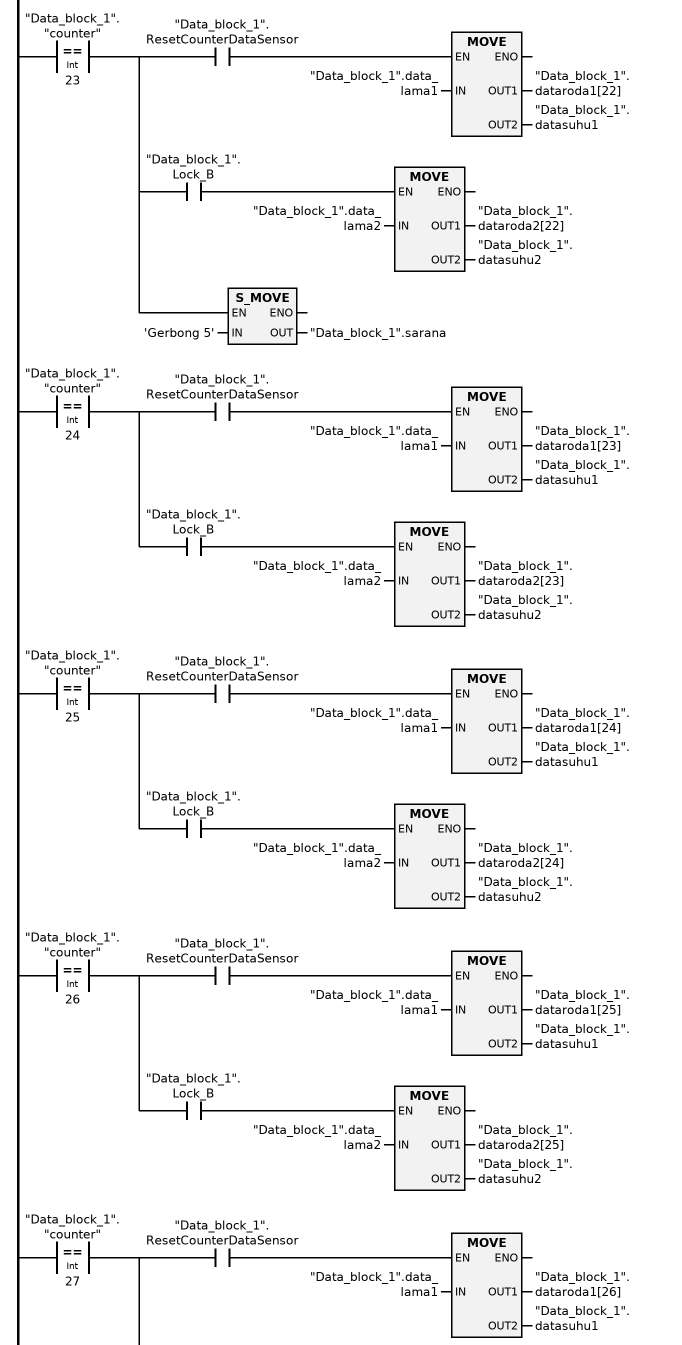
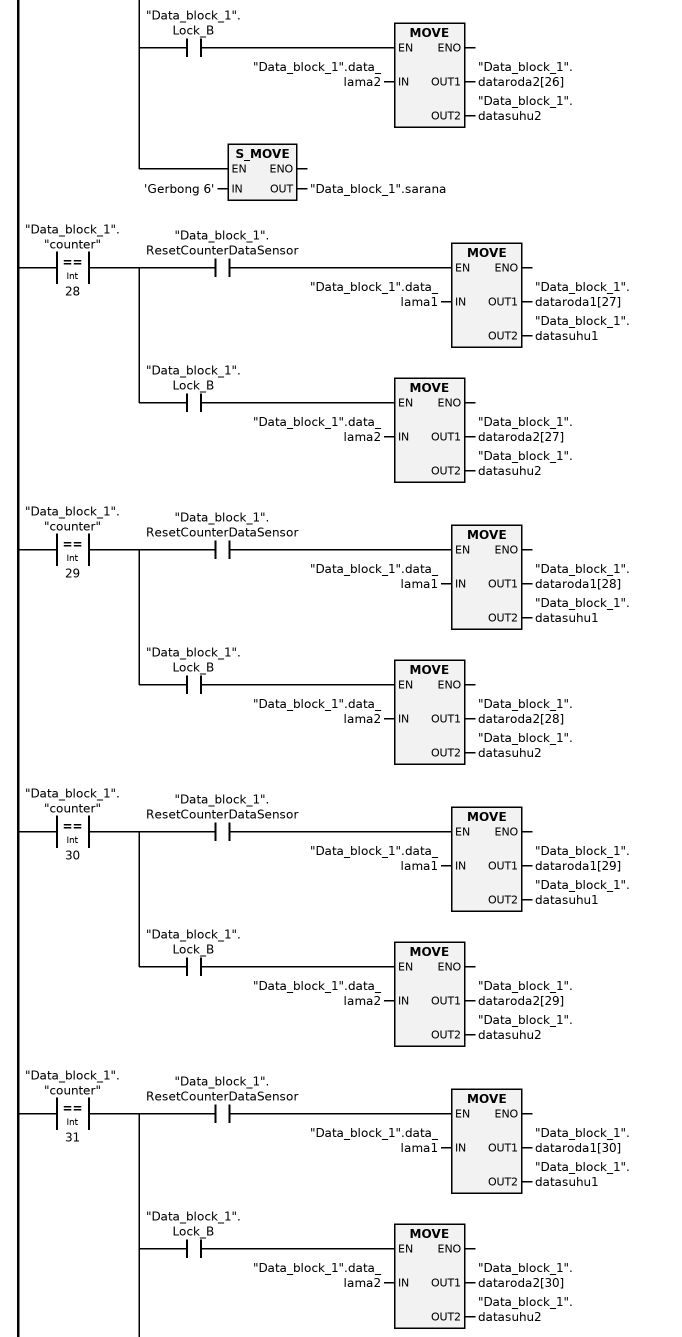
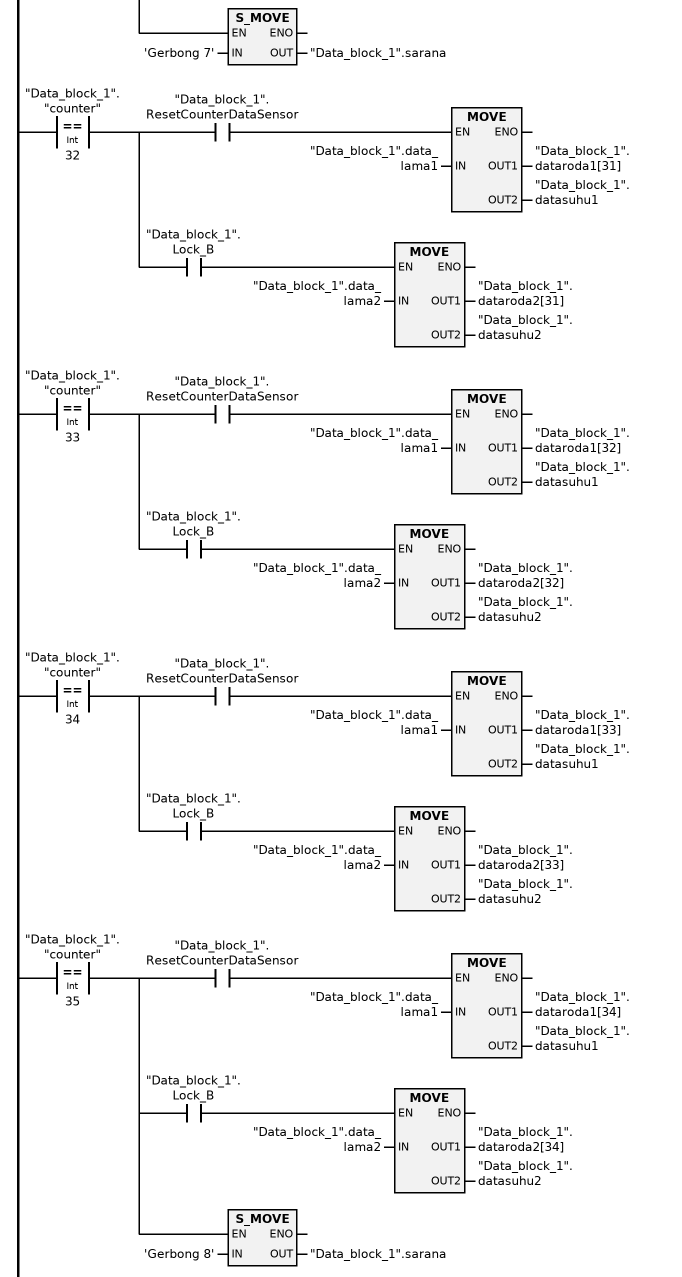
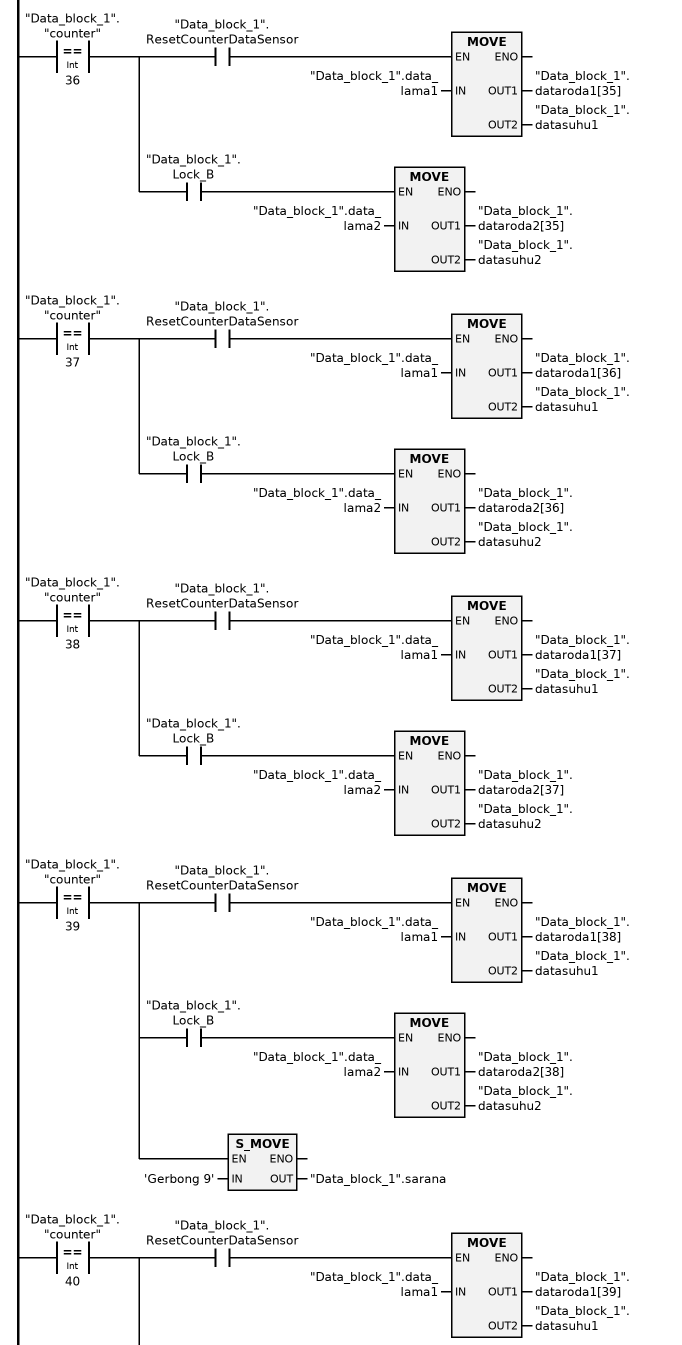
